  Call Extruder(294.14489)
  MoveL 3985 to (558.92, 479.39, 68) mm, rotated rx 180 ry 0 rz 160 deg; joints [3.193, 77.828, -27.011, -151.068, 54.497, 162.203]
  Set speed (17.7 mm/s)
  Call Extruder(298.39452)
  MoveL 3986 to (559.34, 480.66, 68) mm, rotated rx 180 ry 0 rz 160 deg; joints [3.332, 77.936, -27.236, -150.865, 54.438, 162.039]
  Set speed (17.7 mm/s)
  Call Extruder(302.35866)
  MoveL 3987 to (559.73, 481.84, 68) mm, rotated rx 180 ry 0 rz 160 deg; joints [3.463, 78.036, -27.442, -150.675, 54.385, 161.886]
  Call Extruder(306.52683)
  MoveL 3988 to (560.09, 483.1, 68) mm, rotated rx -180 ry 0 rz 160 deg; joints [3.601, 78.133, -27.644, -150.477, 54.338, 161.729]
  Set speed (17.7 mm/s)
  Call Extruder(310.60092)
  MoveL 3989 to (560.43, 484.33, 68) mm, rotated rx 180 ry 0 rz 160 deg; joints [3.736, 78.225, -27.836, -150.283, 54.294, 161.576]
  Set speed (17.7 mm/s)
  Call Extruder(318.62879)
  MoveL 3990 to (561.01, 486.78, 68) mm, rotated rx -180 ry 0 rz 160 deg; joints [4.006, 78.393, -28.184, -149.903, 54.224, 161.281]
  Set speed (17.7 mm/s)
  Call Extruder(326.84459)
  MoveL 3991 to (561.5, 489.31, 68) mm, rotated rx 180 ry 0 rz 160 deg; joints [4.285, 78.545, -28.498, -149.519, 54.173, 160.99]
  Set speed (17.7 mm/s)
  Call Extruder(334.91481)
  MoveL 3992 to (561.89, 491.82, 68) mm, rotated rx -180 ry 0 rz 160 deg; joints [4.561, 78.676, -28.769, -149.146, 54.144, 160.714]
  Set speed (17.7 mm/s)
  Call Extruder(343.20136)
  MoveL 3993 to (562.17, 494.4, 68) mm, rotated rx -180 ry 0 rz 160 deg; joints [4.846, 78.79, -29.004, -148.769, 54.134, 160.442]
  Set speed (17.7 mm/s)
  Call Extruder(351.25389)
  MoveL 3994 to (562.35, 496.93, 68) mm, rotated rx 180 ry 0 rz 160 deg; joints [5.124, 78.88, -29.191, -148.409, 54.146, 160.191]
  Set speed (17.7 mm/s)
  Call Extruder(359.37485)
  MoveL 3995 to (562.42, 499.47, 68) mm, rotated rx -180 ry 0 rz 160 deg; joints [5.407, 78.951, -29.336, -148.053, 54.178, 159.95]
  Set speed (17.7 mm/s)
  Call Extruder(367.60614)
  MoveL 3996 to (562.39, 502.06, 68) mm, rotated rx -180 ry 0 rz 160 deg; joints [5.694, 79.001, -29.441, -147.701, 54.232, 159.721]
  Set speed (17.7 mm/s)
  Call Extruder(375.64241)
  MoveL 3997 to (562.26, 504.58, 68) mm, rotated rx 180 ry 0 rz 160 deg; joints [5.975, 79.03, -29.501, -147.364, 54.304, 159.511]
  Set speed (17.7 mm/s)
  Call Extruder(383.68912)
  MoveL 3998 to (562.02, 507.09, 68) mm, rotated rx 180 ry 0 rz 160 deg; joints [6.256, 79.038, -29.516, -147.037, 54.396, 159.317]
  Set speed (17.7 mm/s)
  Call Extruder(391.74017)
  MoveL 3999 to (561.68, 509.6, 68) mm, rotated rx 180 ry 0 rz 160 deg; joints [6.538, 79.024, -29.487, -146.719, 54.508, 159.138]
  Set speed (17.7 mm/s)
  Call Extruder(400.03241)
  MoveL 4000 to (561.23, 512.16, 68) mm, rotated rx -180 ry 0 rz 160 deg; joints [6.827, 78.989, -29.416, -146.402, 54.643, 158.971]
  Set speed (17.7 mm/s)
  Call Extruder(408.22270)
  MoveL 4001 to (560.67, 514.68, 68) mm, rotated rx 180 ry 0 rz 160 deg; joints [7.113, 78.932, -29.298, -146.099, 54.796, 158.824]
  Set speed (17.7 mm/s)
  Call Extruder(412.26719)
  MoveL 4002 to (560.36, 515.9, 68) mm, rotated rx -180 ry 0 rz 160 deg; joints [7.253, 78.895, -29.222, -145.955, 54.879, 158.758]
  Set speed (17.7 mm/s)
  Call Extruder(416.24101)
  MoveL 4003 to (560.03, 517.11, 68) mm, rotated rx -180 ry 0 rz 160 deg; joints [7.391, 78.857, -29.142, -145.814, 54.963, 158.696]
  Set speed (17.7 mm/s)
  Call Extruder(420.44181)
  MoveL 4004 to (559.65, 518.37, 68) mm, rotated rx -180 ry 0 rz 160 deg; joints [7.536, 78.808, -29.042, -145.67, 55.059, 158.638]
  Call Extruder(424.29152)
  MoveL 4005 to (559.29, 519.52, 68) mm, rotated rx -180 ry 0 rz 160 deg; joints [7.668, 78.761, -28.945, -145.539, 55.148, 158.586]
  Set speed (17.7 mm/s)
  Call Extruder(432.46928)
  MoveL 4006 to (558.44, 521.94, 68) mm, rotated rx -180 ry 0 rz 160 deg; joints [7.949, 78.644, -28.701, -145.27, 55.354, 158.491]
  Set speed (17.7 mm/s)
  Call Extruder(436.67674)
  MoveL 4007 to (557.96, 523.17, 68) mm, rotated rx 180 ry 0 rz 160 deg; joints [8.093, 78.574, -28.558, -145.137, 55.468, 158.451]
  Set speed (17.7 mm/s)
  Call Extruder(440.85646)
  MoveL 4008 to (557.47, 524.38, 68) mm, rotated rx 180 ry 0 rz 160 deg; joints [8.235, 78.503, -28.41, -145.007, 55.583, 158.413]
  Set speed (17.7 mm/s)
  Call Extruder(448.69676)
  MoveL 4009 to (556.46, 526.63, 68) mm, rotated rx 180 ry 0 rz 160 deg; joints [8.5, 78.352, -28.098, -144.771, 55.812, 158.357]
  Set speed (17.7 mm/s)
  Call Extruder(451.96551)
  MoveL 4010 to (556.02, 527.56, 68) mm, rotated rx 180 ry 0 rz 160 deg; joints [8.61, 78.285, -27.959, -144.676, 55.912, 158.338]
  Set speed (17.7 mm/s)
  Call Extruder(459.02585)
  MoveL 4011 to (555, 529.53, 68) mm, rotated rx -180 ry 0 rz 160 deg; joints [8.846, 78.128, -27.634, -144.477, 56.136, 158.307]
  Set speed (17.7 mm/s)
  Call Extruder(465.05663)
  MoveL 4012 to (554.08, 531.18, 68) mm, rotated rx -180 ry 0 rz 160 deg; joints [9.046, 77.983, -27.333, -144.315, 56.337, 158.293]
  Set speed (17.7 mm/s)
  Call Extruder(469.10106)
  MoveL 4013 to (553.43, 532.28, 68) mm, rotated rx 180 ry 0 rz 160 deg; joints [9.179, 77.881, -27.121, -144.209, 56.475, 158.288]
  Set speed (17.7 mm/s)
  Call Extruder(472.62067)
  MoveL 4014 to (552.85, 533.22, 68) mm, rotated rx -180 ry 0 rz 160 deg; joints [9.294, 77.788, -26.929, -144.12, 56.598, 158.287]
  Set speed (17.7 mm/s)
  Call Extruder(477.24876)
  MoveL 4015 to (552.07, 534.44, 68) mm, rotated rx -180 ry 0 rz 160 deg; joints [9.444, 77.662, -26.667, -144.005, 56.764, 158.291]
  Set speed (17.7 mm/s)
  Call Extruder(482.03626)
  MoveL 4016 to (551.22, 535.68, 68) mm, rotated rx -180 ry 0 rz 160 deg; joints [9.598, 77.526, -26.384, -143.89, 56.94, 158.3]
  Set speed (17.7 mm/s)
  Call Extruder(485.47775)
  MoveL 4017 to (550.6, 536.56, 68) mm, rotated rx 180 ry 0 rz 160 deg; joints [9.708, 77.426, -26.175, -143.81, 57.068, 158.31]
  Call Extruder(489.58215)
  MoveL 4018 to (549.83, 537.6, 68) mm, rotated rx -180 ry 0 rz 160 deg; joints [9.838, 77.301, -25.915, -143.718, 57.225, 158.327]
  Call Extruder(493.57157)
  MoveL 4019 to (549.07, 538.59, 68) mm, rotated rx 180 ry 0 rz 160 deg; joints [9.964, 77.176, -25.655, -143.631, 57.38, 158.348]
  Call Extruder(497.29229)
  MoveL 4020 to (548.34, 539.5, 68) mm, rotated rx 180 ry 0 rz 160 deg; joints [10.08, 77.058, -25.408, -143.551, 57.527, 158.369]
  Set speed (17.7 mm/s)
  Call Extruder(501.66302)
  MoveL 4021 to (547.45, 540.56, 68) mm, rotated rx -180 ry 0 rz 160 deg; joints [10.215, 76.914, -25.108, -143.462, 57.702, 158.4]
  Set speed (17.7 mm/s)
  Call Extruder(505.72359)
  MoveL 4022 to (546.62, 541.52, 68) mm, rotated rx -180 ry 0 rz 160 deg; joints [10.339, 76.777, -24.821, -143.381, 57.868, 158.432]
  Call Extruder(509.84035)
  MoveL 4023 to (545.75, 542.47, 68) mm, rotated rx -180 ry 0 rz 160 deg; joints [10.464, 76.634, -24.524, -143.302, 58.038, 158.469]
  Call Extruder(513.86834)
  MoveL 4024 to (544.88, 543.39, 68) mm, rotated rx 180 ry 0 rz 160 deg; joints [10.585, 76.492, -24.226, -143.227, 58.207, 158.508]
  Call Extruder(517.98050)
  MoveL 4025 to (543.97, 544.31, 68) mm, rotated rx 180 ry 0 rz 160 deg; joints [10.707, 76.343, -23.915, -143.154, 58.382, 158.553]
  Set speed (17.7 mm/s)
  Call Extruder(522.01486)
  MoveL 4026 to (543.06, 545.19, 68) mm, rotated rx -180 ry 0 rz 160 deg; joints [10.826, 76.194, -23.602, -143.085, 58.556, 158.6]
  Set speed (17.7 mm/s)
  Call Extruder(526.03664)
  MoveL 4027 to (542.14, 546.05, 68) mm, rotated rx -180 ry 0 rz 160 deg; joints [10.942, 76.043, -23.286, -143.018, 58.731, 158.65]
  Set speed (17.7 mm/s)
  Call Extruder(530.16740)
  MoveL 4028 to (541.17, 546.92, 68) mm, rotated rx 180 ry 0 rz 160 deg; joints [11.061, 75.885, -22.954, -142.953, 58.913, 158.706]
  Set speed (17.7 mm/s)
  Call Extruder(534.20745)
  MoveL 4029 to (540.21, 547.75, 68) mm, rotated rx 180 ry 0 rz 160 deg; joints [11.175, 75.728, -22.623, -142.891, 59.092, 158.764]
  Call Extruder(538.24993)
  MoveL 4030 to (539.23, 548.55, 68) mm, rotated rx -180 ry 0 rz 160 deg; joints [11.288, 75.568, -22.286, -142.832, 59.274, 158.825]
  Set speed (17.7 mm/s)
  Call Extruder(542.31774)
  MoveL 4031 to (538.23, 549.35, 68) mm, rotated rx 180 ry 0 rz 160 deg; joints [11.4, 75.404, -21.942, -142.775, 59.459, 158.89]
  Set speed (17.7 mm/s)
  Call Extruder(546.38760)
  MoveL 4032 to (537.21, 550.12, 68) mm, rotated rx 180 ry 0 rz 160 deg; joints [11.511, 75.238, -21.592, -142.721, 59.645, 158.959]
  Set speed (17.7 mm/s)
  Call Extruder(550.65806)
  MoveL 4033 to (536.13, 550.91, 68) mm, rotated rx -180 ry 0 rz 160 deg; joints [11.625, 75.062, -21.22, -142.667, 59.842, 159.034]
  Call Extruder(554.55663)
  MoveL 4034 to (535.12, 551.61, 68) mm, rotated rx 180 ry 0 rz 160 deg; joints [11.728, 74.899, -20.875, -142.619, 60.023, 159.106]
  Set speed (17.7 mm/s)
  Call Extruder(558.59833)
  MoveL 4035 to (534.07, 552.31, 68) mm, rotated rx 180 ry 0 rz 160 deg; joints [11.833, 74.727, -20.512, -142.573, 60.212, 159.184]
  Set speed (17.7 mm/s)
  Call Extruder(562.67182)
  MoveL 4036 to (532.99, 553, 68) mm, rotated rx 180 ry 0 rz 160 deg; joints [11.937, 74.552, -20.142, -142.529, 60.404, 159.265]
  Set speed (17.7 mm/s)
  Call Extruder(566.75852)
  MoveL 4037 to (531.89, 553.66, 68) mm, rotated rx 180 ry 0 rz 160 deg; joints [12.039, 74.375, -19.767, -142.488, 60.597, 159.349]
  Set speed (17.7 mm/s)
  Call Extruder(570.85954)
  MoveL 4038 to (530.78, 554.31, 68) mm, rotated rx -180 ry 0 rz 160 deg; joints [12.14, 74.196, -19.386, -142.448, 60.793, 159.437]
  Set speed (17.7 mm/s)
  Call Extruder(576.98550)
  MoveL 4039 to (529.09, 555.24, 68) mm, rotated rx -180 ry 0 rz 160 deg; joints [12.288, 73.925, -18.81, -142.393, 61.086, 159.573]
  Call Extruder(583.05688)
  MoveL 4040 to (527.39, 556.1, 68) mm, rotated rx 180 ry 0 rz 160 deg; joints [12.429, 73.652, -18.229, -142.346, 61.379, 159.715]
  Set speed (17.7 mm/s)
  Call Extruder(587.00755)
  MoveL 4041 to (526.27, 556.63, 68) mm, rotated rx -180 ry 0 rz 160 deg; joints [12.519, 73.473, -17.847, -142.317, 61.571, 159.81]
  Set speed (17.7 mm/s)
  Call Extruder(591.18449)
  MoveL 4042 to (525.07, 557.16, 68) mm, rotated rx -180 ry 0 rz 160 deg; joints [12.61, 73.282, -17.44, -142.29, 61.774, 159.914]
  Set speed (17.7 mm/s)
  Call Extruder(595.25468)
  MoveL 4043 to (523.9, 557.67, 68) mm, rotated rx -180 ry 0 rz 160 deg; joints [12.699, 73.096, -17.042, -142.265, 61.971, 160.016]
  Call Extruder(599.32932)
  MoveL 4044 to (522.71, 558.14, 68) mm, rotated rx 180 ry 0 rz 160 deg; joints [12.784, 72.908, -16.639, -142.244, 62.17, 160.123]
  Set speed (17.7 mm/s)
  Call Extruder(603.41760)
  MoveL 4045 to (521.51, 558.6, 68) mm, rotated rx -180 ry 0 rz 160 deg; joints [12.869, 72.719, -16.234, -142.224, 62.37, 160.231]
  Set speed (17.7 mm/s)
  Call Extruder(607.51619)
  MoveL 4046 to (520.3, 559.02, 68) mm, rotated rx 180 ry 0 rz 160 deg; joints [12.95, 72.527, -15.823, -142.208, 62.571, 160.342]
  Set speed (17.7 mm/s)
  Call Extruder(611.50972)
  MoveL 4047 to (519.11, 559.43, 68) mm, rotated rx 180 ry 0 rz 160 deg; joints [13.029, 72.341, -15.423, -142.192, 62.766, 160.452]
  Set speed (17.7 mm/s)
  Call Extruder(615.60966)
  MoveL 4048 to (517.88, 559.8, 68) mm, rotated rx -180 ry 0 rz 160 deg; joints [13.105, 72.148, -15.007, -142.181, 62.968, 160.568]
  Call Extruder(619.63022)
  MoveL 4049 to (516.67, 560.16, 68) mm, rotated rx 180 ry 0 rz 160 deg; joints [13.18, 71.959, -14.6, -142.171, 63.165, 160.683]
  Set speed (17.7 mm/s)
  Call Extruder(623.21774)
  MoveL 4050 to (515.59, 560.44, 68) mm, rotated rx -180 ry 0 rz 160 deg; joints [13.243, 71.79, -14.233, -142.165, 63.341, 160.788]
  Call Extruder(627.77646)
  MoveL 4051 to (514.2, 560.79, 68) mm, rotated rx -180 ry 0 rz 160 deg; joints [13.321, 71.574, -13.768, -142.158, 63.564, 160.922]
  Set speed (17.7 mm/s)
  Call Extruder(635.96464)
  MoveL 4052 to (511.68, 561.32, 68) mm, rotated rx 180 ry 0 rz 160 deg; joints [13.454, 71.185, -12.924, -142.156, 63.966, 161.171]
  Set speed (17.7 mm/s)
  Call Extruder(644.15315)
  MoveL 4053 to (509.15, 561.75, 68) mm, rotated rx 180 ry 0 rz 160 deg; joints [13.576, 70.795, -12.077, -142.163, 64.367, 161.427]
  Set speed (17.7 mm/s)
  Call Extruder(652.20654)
  MoveL 4054 to (506.64, 562.07, 68) mm, rotated rx 180 ry 0 rz 160 deg; joints [13.686, 70.411, -11.24, -142.179, 64.759, 161.685]
  Set speed (17.7 mm/s)
  Call Extruder(660.39241)
  MoveL 4055 to (504.08, 562.29, 68) mm, rotated rx -180 ry 0 rz 160 deg; joints [13.787, 70.021, -10.386, -142.207, 65.157, 161.954]
  Set speed (17.7 mm/s)
  Call Extruder(668.57383)
  MoveL 4056 to (501.52, 562.4, 68) mm, rotated rx 180 ry 0 rz 160 deg; joints [13.876, 69.632, -9.533, -142.244, 65.551, 162.228]
  Set speed (17.7 mm/s)
  Call Extruder(676.52907)
  MoveL 4057 to (499.02, 562.42, 68) mm, rotated rx 180 ry 0 rz 160 deg; joints [13.952, 69.256, -8.704, -142.289, 65.932, 162.499]
  Set speed (10.0 mm/s)
  MoveL 4058 to (499.02, 562.42, 72) mm, rotated rx 180 ry 0 rz 160 deg; joints [13.952, 68.584, -8.319, -142.211, 65.706, 162.307]
  Set speed (120.0 mm/s)
  MoveL 4059 to (498.98, 563.11, 72) mm, rotated rx 180 ry 0 rz 160 deg; joints [14.037, 68.604, -8.362, -142.116, 65.713, 162.255]
  Set speed (17.8 mm/s)
  Call Extruder(684.78584)
  MoveL 4060 to (496.38, 563.01, 72) mm, rotated rx 180 ry 0 rz 160 deg; joints [14.103, 68.213, -7.503, -142.174, 66.103, 162.541]
  Set speed (17.7 mm/s)
  Call Extruder(693.01751)
  MoveL 4061 to (493.8, 562.81, 72) mm, rotated rx 180 ry 0 rz 160 deg; joints [14.158, 67.826, -6.651, -142.243, 66.487, 162.83]
  Set speed (17.8 mm/s)
  Call Extruder(701.15810)
  MoveL 4062 to (491.26, 562.51, 72) mm, rotated rx 180 ry 0 rz 160 deg; joints [14.199, 67.447, -5.811, -142.321, 66.863, 163.119]
  Set speed (17.8 mm/s)
  Call Extruder(709.32825)
  MoveL 4063 to (488.72, 562.1, 72) mm, rotated rx 180 ry 0 rz 160 deg; joints [14.228, 67.07, -4.974, -142.411, 67.236, 163.413]
  Call Extruder(717.38257)
  MoveL 4064 to (486.24, 561.6, 72) mm, rotated rx -180 ry 0 rz 160 deg; joints [14.243, 66.702, -4.155, -142.509, 67.598, 163.705]
  Set speed (17.7 mm/s)
  Call Extruder(721.73346)
  MoveL 4065 to (484.9, 561.28, 72) mm, rotated rx 180 ry 0 rz 160 deg; joints [14.246, 66.506, -3.716, -142.567, 67.791, 163.863]
  Set speed (17.7 mm/s)
  Call Extruder(725.73905)
  MoveL 4066 to (483.69, 560.97, 72) mm, rotated rx -180 ry 0 rz 160 deg; joints [14.246, 66.326, -3.314, -142.621, 67.968, 164.008]
  Call Extruder(729.90744)
  MoveL 4067 to (482.43, 560.62, 72) mm, rotated rx 180 ry 0 rz 160 deg; joints [14.242, 66.14, -2.898, -142.682, 68.15, 164.161]
  Set speed (17.7 mm/s)
  Call Extruder(734.10375)
  MoveL 4068 to (481.16, 560.24, 72) mm, rotated rx 180 ry 0 rz 160 deg; joints [14.235, 65.955, -2.481, -142.745, 68.332, 164.314]
  Set speed (17.7 mm/s)
  Call Extruder(738.10997)
  MoveL 4069 to (479.97, 559.85, 72) mm, rotated rx 180 ry 0 rz 160 deg; joints [14.223, 65.779, -2.086, -142.809, 68.504, 164.462]
  Set speed (17.7 mm/s)
  Call Extruder(742.27099)
  MoveL 4070 to (478.73, 559.43, 72) mm, rotated rx 180 ry 0 rz 160 deg; joints [14.21, 65.598, -1.678, -142.877, 68.681, 164.614]
  Set speed (17.7 mm/s)
  Call Extruder(746.37719)
  MoveL 4071 to (477.52, 558.97, 72) mm, rotated rx 180 ry 0 rz 160 deg; joints [14.191, 65.421, -1.278, -142.949, 68.854, 164.765]
  Call Extruder(750.35027)
  MoveL 4072 to (476.36, 558.52, 72) mm, rotated rx 180 ry 0 rz 160 deg; joints [14.172, 65.251, -0.893, -143.019, 69.02, 164.911]
  Set speed (17.7 mm/s)
  Call Extruder(752.50038)
  MoveL 4073 to (475.73, 558.27, 72) mm, rotated rx 180 ry 0 rz 160 deg; joints [14.159, 65.16, -0.687, -143.058, 69.109, 164.99]
  Set speed (17.7 mm/s)
  Call Extruder(758.47349)
  MoveL 4074 to (474.01, 557.52, 72) mm, rotated rx 180 ry 0 rz 160 deg; joints [14.119, 64.909, -0.117, -143.172, 69.354, 165.209]
  Set speed (17.8 mm/s)
  Call Extruder(762.73063)
  MoveL 4075 to (472.8, 556.95, 72) mm, rotated rx -180 ry 0 rz 160 deg; joints [14.086, 64.732, 0.286, -143.257, 69.527, 165.366]
  Call Extruder(766.79294)
  MoveL 4076 to (471.65, 556.39, 72) mm, rotated rx 180 ry 0 rz 160 deg; joints [14.051, 64.565, 0.667, -143.341, 69.689, 165.515]
  Set speed (17.7 mm/s)
  Call Extruder(769.82727)
  MoveL 4077 to (470.8, 555.96, 72) mm, rotated rx -180 ry 0 rz 160 deg; joints [14.023, 64.442, 0.949, -143.405, 69.81, 165.626]
  Set speed (17.7 mm/s)
  Call Extruder(775.14653)
  MoveL 4078 to (469.33, 555.16, 72) mm, rotated rx 180 ry 0 rz 160 deg; joints [13.968, 64.228, 1.439, -143.522, 70.018, 165.82]
  Set speed (17.8 mm/s)
  Call Extruder(779.12231)
  MoveL 4079 to (468.24, 554.54, 72) mm, rotated rx 180 ry 0 rz 160 deg; joints [13.923, 64.07, 1.801, -143.612, 70.171, 165.965]
  Set speed (17.8 mm/s)
  Call Extruder(783.32191)
  MoveL 4080 to (467.11, 553.87, 72) mm, rotated rx -180 ry 0 rz 160 deg; joints [13.871, 63.905, 2.18, -143.711, 70.331, 166.118]
  Set speed (17.8 mm/s)
  Call Extruder(787.31436)
  MoveL 4081 to (466.04, 553.2, 72) mm, rotated rx 180 ry 0 rz 160 deg; joints [13.819, 63.75, 2.536, -143.807, 70.481, 166.262]
  Set speed (17.8 mm/s)
  Call Extruder(791.45586)
  MoveL 4082 to (464.95, 552.49, 72) mm, rotated rx -180 ry 0 rz 160 deg; joints [13.761, 63.592, 2.901, -143.91, 70.634, 166.411]
  Set speed (17.8 mm/s)
  Call Extruder(795.56231)
  MoveL 4083 to (463.88, 551.76, 72) mm, rotated rx -180 ry 0 rz 160 deg; joints [13.7, 63.437, 3.259, -144.015, 70.784, 166.559]
  Set speed (17.8 mm/s)
  Call Extruder(799.66580)
  MoveL 4084 to (462.83, 551.01, 72) mm, rotated rx -180 ry 0 rz 160 deg; joints [13.635, 63.285, 3.613, -144.122, 70.932, 166.705]
  Set speed (17.7 mm/s)
  Call Extruder(803.84529)
  MoveL 4085 to (461.78, 550.23, 72) mm, rotated rx -180 ry 0 rz 160 deg; joints [13.566, 63.132, 3.968, -144.235, 71.08, 166.854]
  Set speed (17.7 mm/s)
  Call Extruder(807.89672)
  MoveL 4086 to (460.77, 549.45, 72) mm, rotated rx 180 ry 0 rz 160 deg; joints [13.494, 62.986, 4.308, -144.346, 71.221, 166.997]
  Set speed (17.8 mm/s)
  Call Extruder(812.15374)
  MoveL 4087 to (459.73, 548.6, 72) mm, rotated rx 180 ry 0 rz 160 deg; joints [13.416, 62.834, 4.66, -144.467, 71.367, 167.146]
  Call Extruder(816.08698)
  MoveL 4088 to (458.79, 547.8, 72) mm, rotated rx 180 ry 0 rz 160 deg; joints [13.339, 62.697, 4.98, -144.581, 71.499, 167.284]
  Call Extruder(820.12043)
  MoveL 4089 to (457.83, 546.96, 72) mm, rotated rx -180 ry 0 rz 160 deg; joints [13.258, 62.558, 5.305, -144.701, 71.633, 167.423]
  Set speed (17.8 mm/s)
  Call Extruder(824.28360)
  MoveL 4090 to (456.87, 546.08, 72) mm, rotated rx 180 ry 0 rz 160 deg; joints [13.17, 62.418, 5.634, -144.827, 71.768, 167.567]
  Set speed (17.8 mm/s)
  Call Extruder(828.39151)
  MoveL 4091 to (455.93, 545.19, 72) mm, rotated rx 180 ry 0 rz 160 deg; joints [13.079, 62.282, 5.954, -144.955, 71.899, 167.707]
  Call Extruder(832.47818)
  MoveL 4092 to (455.02, 544.28, 72) mm, rotated rx -180 ry 0 rz 160 deg; joints [12.986, 62.149, 6.267, -145.085, 72.027, 167.845]
  Set speed (17.8 mm/s)
  Call Extruder(836.60977)
  MoveL 4093 to (454.12, 543.34, 72) mm, rotated rx -180 ry 0 rz 160 deg; joints [12.888, 62.017, 6.578, -145.219, 72.153, 167.983]
  Set speed (17.8 mm/s)
  Call Extruder(840.62722)
  MoveL 4094 to (453.26, 542.42, 72) mm, rotated rx 180 ry 0 rz 160 deg; joints [12.789, 61.891, 6.875, -145.351, 72.273, 168.117]
  Call Extruder(844.81137)
  MoveL 4095 to (452.39, 541.43, 72) mm, rotated rx -180 ry 0 rz 160 deg; joints [12.682, 61.763, 7.178, -145.493, 72.396, 168.255]
  Call Extruder(848.43498)
  MoveL 4096 to (451.65, 540.57, 72) mm, rotated rx -180 ry 0 rz 160 deg; joints [12.587, 61.654, 7.436, -145.617, 72.499, 168.373]
  Set speed (17.8 mm/s)
  Call Extruder(853.01287)
  MoveL 4097 to (450.73, 539.45, 72) mm, rotated rx -180 ry 0 rz 160 deg; joints [12.463, 61.519, 7.756, -145.778, 72.627, 168.52]
  Call Extruder(857.11960)
  MoveL 4098 to (449.94, 538.43, 72) mm, rotated rx 180 ry 0 rz 160 deg; joints [12.348, 61.402, 8.036, -145.924, 72.739, 168.651]
  Set speed (17.8 mm/s)
  Call Extruder(861.20079)
  MoveL 4099 to (449.16, 537.41, 72) mm, rotated rx 180 ry 0 rz 160 deg; joints [12.23, 61.287, 8.309, -146.072, 72.847, 168.779]
  Call Extruder(865.32794)
  MoveL 4100 to (448.4, 536.36, 72) mm, rotated rx 180 ry 0 rz 160 deg; joints [12.108, 61.174, 8.578, -146.225, 72.954, 168.907]
  Call Extruder(869.40800)
  MoveL 4101 to (447.68, 535.3, 72) mm, rotated rx 180 ry 0 rz 160 deg; joints [11.983, 61.065, 8.838, -146.378, 73.056, 169.033]
  Set speed (17.8 mm/s)
  Call Extruder(873.51158)
  MoveL 4102 to (446.97, 534.22, 72) mm, rotated rx 180 ry 0 rz 160 deg; joints [11.855, 60.959, 9.094, -146.535, 73.156, 169.157]
  Set speed (17.8 mm/s)
  Call Extruder(877.62154)
  MoveL 4103 to (446.27, 533.13, 72) mm, rotated rx 180 ry 0 rz 160 deg; joints [11.723, 60.855, 9.344, -146.694, 73.253, 169.279]
  Set speed (17.8 mm/s)
  Call Extruder(881.67014)
  MoveL 4104 to (445.62, 532.04, 72) mm, rotated rx -180 ry 0 rz 160 deg; joints [11.591, 60.755, 9.583, -146.853, 73.345, 169.399]
  Call Extruder(885.83166)
  MoveL 4105 to (444.96, 530.9, 72) mm, rotated rx -180 ry 0 rz 160 deg; joints [11.451, 60.656, 9.822, -147.019, 73.437, 169.519]
  Call Extruder(889.93873)
  MoveL 4106 to (444.35, 529.77, 72) mm, rotated rx 180 ry 0 rz 160 deg; joints [11.31, 60.561, 10.051, -147.186, 73.524, 169.636]
  Call Extruder(894.04948)
  MoveL 4107 to (443.75, 528.62, 72) mm, rotated rx 180 ry 0 rz 160 deg; joints [11.166, 60.469, 10.274, -147.354, 73.608, 169.752]
  Set speed (17.8 mm/s)
  Call Extruder(898.06498)
  MoveL 4108 to (443.18, 527.49, 72) mm, rotated rx -180 ry 0 rz 160 deg; joints [11.022, 60.382, 10.485, -147.521, 73.687, 169.862]
  Set speed (17.7 mm/s)
  Call Extruder(902.33645)
  MoveL 4109 to (442.62, 526.27, 72) mm, rotated rx -180 ry 0 rz 160 deg; joints [10.866, 60.293, 10.7, -147.701, 73.766, 169.978]
  Set speed (17.7 mm/s)
  Call Extruder(906.43110)
  MoveL 4110 to (442.09, 525.1, 72) mm, rotated rx -180 ry 0 rz 160 deg; joints [10.715, 60.21, 10.902, -147.874, 73.84, 170.087]
  Set speed (17.7 mm/s)
  Call Extruder(910.55447)
  MoveL 4111 to (441.59, 523.9, 72) mm, rotated rx -180 ry 0 rz 160 deg; joints [10.559, 60.13, 11.096, -148.052, 73.91, 170.194]
  Set speed (17.7 mm/s)
  Call Extruder(914.45439)
  MoveL 4112 to (441.13, 522.77, 72) mm, rotated rx 180 ry 0 rz 160 deg; joints [10.41, 60.057, 11.274, -148.221, 73.975, 170.295]
  Set speed (17.7 mm/s)
  Call Extruder(918.77421)
  MoveL 4113 to (440.66, 521.5, 72) mm, rotated rx -180 ry 0 rz 160 deg; joints [10.241, 59.98, 11.462, -148.41, 74.04, 170.403]
  Call Extruder(922.87536)
  MoveL 4114 to (440.23, 520.28, 72) mm, rotated rx 180 ry 0 rz 160 deg; joints [10.08, 59.908, 11.636, -148.591, 74.101, 170.504]
  Set speed (17.8 mm/s)
  Call Extruder(931.08749)
  MoveL 4115 to (439.45, 517.82, 72) mm, rotated rx 180 ry 0 rz 160 deg; joints [9.747, 59.777, 11.958, -148.96, 74.21, 170.7]
  Set speed (17.7 mm/s)
  Call Extruder(935.19094)
  MoveL 4116 to (439.11, 516.58, 72) mm, rotated rx 180 ry 0 rz 160 deg; joints [9.578, 59.716, 12.106, -149.147, 74.257, 170.794]
  Set speed (17.7 mm/s)
  Call Extruder(939.16372)
  MoveL 4117 to (438.79, 515.37, 72) mm, rotated rx 180 ry 0 rz 160 deg; joints [9.412, 59.66, 12.245, -149.328, 74.302, 170.883]
  Set speed (17.7 mm/s)
  Call Extruder(943.40434)
  MoveL 4118 to (438.48, 514.07, 72) mm, rotated rx 180 ry 0 rz 160 deg; joints [9.233, 59.604, 12.382, -149.524, 74.344, 170.976]
  Call Extruder(947.41026)
  MoveL 4119 to (438.2, 512.85, 72) mm, rotated rx 180 ry 0 rz 160 deg; joints [9.062, 59.552, 12.508, -149.71, 74.381, 171.062]
  Set speed (17.8 mm/s)
  Call Extruder(955.74907)
  MoveL 4120 to (437.72, 510.27, 72) mm, rotated rx -180 ry 0 rz 160 deg; joints [8.701, 59.457, 12.742, -150.1, 74.446, 171.234]
  Set speed (17.7 mm/s)
  Call Extruder(963.95051)
  MoveL 4121 to (437.36, 507.71, 72) mm, rotated rx 180 ry 0 rz 160 deg; joints [8.339, 59.377, 12.94, -150.487, 74.494, 171.394]
  Call Extruder(972.16130)
  MoveL 4122 to (437.1, 505.15, 72) mm, rotated rx 180 ry 0 rz 160 deg; joints [7.971, 59.309, 13.107, -150.878, 74.526, 171.546]
  Call Extruder(980.19898)
  MoveL 4123 to (436.94, 502.62, 72) mm, rotated rx 180 ry 0 rz 160 deg; joints [7.607, 59.255, 13.24, -151.263, 74.542, 171.685]
  Set speed (17.7 mm/s)
  Call Extruder(988.50118)
  MoveL 4124 to (436.88, 500.01, 72) mm, rotated rx 180 ry 0 rz 160 deg; joints [7.227, 59.213, 13.344, -151.661, 74.542, 171.82]
  Call Extruder(995.96639)
  MoveL 4125 to (436.93, 497.66, 72) mm, rotated rx -180 ry 0 rz 160 deg; joints [6.883, 59.187, 13.41, -152.019, 74.528, 171.933]
  Call Extruder(1003.17441)
  MoveL 4126 to (437.05, 495.4, 72) mm, rotated rx 180 ry 0 rz 160 deg; joints [6.55, 59.172, 13.447, -152.364, 74.501, 172.035]
  Call Extruder(1010.66998)
  MoveL 4127 to (437.27, 493.06, 72) mm, rotated rx 180 ry 0 rz 160 deg; joints [6.203, 59.167, 13.459, -152.722, 74.459, 172.134]
  Call Extruder(1018.05787)
  MoveL 4128 to (437.56, 490.75, 72) mm, rotated rx -180 ry 0 rz 160 deg; joints [5.861, 59.173, 13.445, -153.073, 74.405, 172.225]
  Set speed (17.7 mm/s)
  Call Extruder(1025.53388)
  MoveL 4129 to (437.95, 488.43, 72) mm, rotated rx 180 ry 0 rz 160 deg; joints [5.515, 59.189, 13.403, -153.425, 74.337, 172.309]
  Set speed (17.8 mm/s)
  Call Extruder(1032.83144)
  MoveL 4130 to (438.41, 486.18, 72) mm, rotated rx 180 ry 0 rz 160 deg; joints [5.179, 59.216, 13.337, -153.766, 74.257, 172.384]
  Call Extruder(1040.21403)
  MoveL 4131 to (438.96, 483.93, 72) mm, rotated rx 180 ry 0 rz 160 deg; joints [4.841, 59.254, 13.243, -154.107, 74.162, 172.453]
  Call Extruder(1047.50290)
  MoveL 4132 to (439.59, 481.72, 72) mm, rotated rx -180 ry 0 rz 160 deg; joints [4.511, 59.302, 13.125, -154.44, 74.055, 172.515]
  Set speed (17.8 mm/s)
  Call Extruder(1054.91227)
  MoveL 4133 to (440.31, 479.5, 72) mm, rotated rx 180 ry 0 rz 160 deg; joints [4.178, 59.361, 12.979, -154.772, 73.934, 172.571]
  Set speed (17.8 mm/s)
  Call Extruder(1062.45704)
  MoveL 4134 to (441.12, 477.27, 72) mm, rotated rx 180 ry 0 rz 160 deg; joints [3.843, 59.432, 12.803, -155.105, 73.796, 172.621]
  Set speed (17.8 mm/s)
  Call Extruder(1069.84361)
  MoveL 4135 to (441.99, 475.12, 72) mm, rotated rx 180 ry 0 rz 160 deg; joints [3.521, 59.512, 12.606, -155.424, 73.648, 172.663]
  Set speed (17.8 mm/s)
  Call Extruder(1077.06733)
  MoveL 4136 to (442.93, 473.05, 72) mm, rotated rx 180 ry 0 rz 160 deg; joints [3.211, 59.601, 12.389, -155.728, 73.491, 172.698]
  Set speed (17.8 mm/s)
  Call Extruder(1084.52838)
  MoveL 4137 to (443.97, 470.94, 72) mm, rotated rx 180 ry 0 rz 160 deg; joints [2.897, 59.703, 12.139, -156.035, 73.316, 172.728]
  Set speed (17.7 mm/s)
  Call Extruder(1091.84400)
  MoveL 4138 to (445.07, 468.92, 72) mm, rotated rx -180 ry 0 rz 160 deg; joints [2.595, 59.813, 11.87, -156.328, 73.132, 172.751]
  Call Extruder(1099.24095)
  MoveL 4139 to (446.25, 466.92, 72) mm, rotated rx 180 ry 0 rz 160 deg; joints [2.298, 59.934, 11.573, -156.615, 72.934, 172.768]
  Set speed (17.8 mm/s)
  Call Extruder(1106.68812)
  MoveL 4140 to (447.51, 464.94, 72) mm, rotated rx -180 ry 0 rz 160 deg; joints [2.006, 60.067, 11.25, -156.895, 72.722, 172.778]
  Set speed (17.8 mm/s)
  Call Extruder(1114.06686)
  MoveL 4141 to (448.84, 463.04, 72) mm, rotated rx -180 ry 0 rz 160 deg; joints [1.726, 60.208, 10.907, -157.162, 72.501, 172.783]
  Call Extruder(1121.45273)
  MoveL 4142 to (450.23, 461.18, 72) mm, rotated rx 180 ry 0 rz 160 deg; joints [1.453, 60.359, 10.539, -157.419, 72.267, 172.781]
  Set speed (17.8 mm/s)
  Call Extruder(1128.76650)
  MoveL 4143 to (451.68, 459.39, 72) mm, rotated rx 180 ry 0 rz 160 deg; joints [1.193, 60.519, 10.153, -157.663, 72.026, 172.774]
  Set speed (17.8 mm/s)
  Call Extruder(1136.30058)
  MoveL 4144 to (453.24, 457.61, 72) mm, rotated rx 180 ry 0 rz 160 deg; joints [0.934, 60.693, 9.733, -157.903, 71.765, 172.76]
  Set speed (17.8 mm/s)
  Call Extruder(1143.69286)
  MoveL 4145 to (454.83, 455.91, 72) mm, rotated rx -180 ry 0 rz 160 deg; joints [0.69, 60.874, 9.299, -158.126, 71.499, 172.74]
  Call Extruder(1150.92671)
  MoveL 4146 to (456.45, 454.31, 72) mm, rotated rx 180 ry 0 rz 160 deg; joints [0.462, 61.059, 8.853, -158.332, 71.229, 172.715]
  Set speed (17.8 mm/s)
  Call Extruder(1158.37668)
  MoveL 4147 to (458.18, 452.73, 72) mm, rotated rx 180 ry 0 rz 160 deg; joints [0.237, 61.26, 8.374, -158.533, 70.941, 172.683]
  Call Extruder(1165.83726)
  MoveL 4148 to (459.97, 451.2, 72) mm, rotated rx -180 ry 0 rz 160 deg; joints [0.023, 61.47, 7.874, -158.721, 70.644, 172.645]
  Call Extruder(1173.08996)
  MoveL 4149 to (461.76, 449.79, 72) mm, rotated rx 180 ry 0 rz 160 deg; joints [-0.175, 61.683, 7.368, -158.891, 70.345, 172.602]
  Set speed (17.8 mm/s)
  Call Extruder(1180.53960)
  MoveL 4150 to (463.65, 448.4, 72) mm, rotated rx -180 ry 0 rz 160 deg; joints [-0.366, 61.91, 6.83, -159.053, 70.031, 172.552]
  Set speed (17.8 mm/s)
  Call Extruder(1187.91519)
  MoveL 4151 to (465.57, 447.1, 72) mm, rotated rx -180 ry 0 rz 160 deg; joints [-0.544, 62.143, 6.279, -159.2, 69.711, 172.496]
  Set speed (17.8 mm/s)
  Call Extruder(1195.37483)
  MoveL 4152 to (467.56, 445.86, 72) mm, rotated rx 180 ry 0 rz 160 deg; joints [-0.713, 62.388, 5.704, -159.334, 69.38, 172.433]
  Call Extruder(1202.76870)
  MoveL 4153 to (469.58, 444.7, 72) mm, rotated rx 180 ry 0 rz 160 deg; joints [-0.868, 62.639, 5.117, -159.454, 69.044, 172.365]
  Set speed (17.8 mm/s)
  Call Extruder(1210.14744)
  MoveL 4154 to (471.63, 443.62, 72) mm, rotated rx -180 ry 0 rz 160 deg; joints [-1.011, 62.896, 4.516, -159.559, 68.703, 172.291]
  Set speed (17.7 mm/s)
  Call Extruder(1217.35488)
  MoveL 4155 to (473.68, 442.64, 72) mm, rotated rx 180 ry 0 rz 160 deg; joints [-1.139, 63.155, 3.913, -159.648, 68.364, 172.212]
  Set speed (17.7 mm/s)
  Call Extruder(1224.66217)
  MoveL 4156 to (475.78, 441.72, 72) mm, rotated rx -180 ry 0 rz 160 deg; joints [-1.257, 63.425, 3.288, -159.725, 68.014, 172.126]
  Set speed (17.8 mm/s)
  Call Extruder(1232.15640)
  MoveL 4157 to (477.97, 440.85, 72) mm, rotated rx -180 ry 0 rz 160 deg; joints [-1.366, 63.709, 2.632, -159.79, 67.65, 172.031]
  Call Extruder(1239.70404)
  MoveL 4158 to (480.21, 440.06, 72) mm, rotated rx -180 ry 0 rz 160 deg; joints [-1.464, 64.002, 1.958, -159.84, 67.279, 171.929]
  Call Extruder(1246.94387)
  MoveL 4159 to (482.39, 439.39, 72) mm, rotated rx -180 ry 0 rz 160 deg; joints [-1.546, 64.289, 1.298, -159.874, 66.918, 171.824]
  Set speed (17.8 mm/s)
  Call Extruder(1254.37889)
  MoveL 4160 to (484.65, 438.78, 72) mm, rotated rx -180 ry 0 rz 160 deg; joints [-1.619, 64.591, 0.609, -159.895, 66.543, 171.71]
  Set speed (17.8 mm/s)
  Call Extruder(1261.85377)
  MoveL 4161 to (486.94, 438.25, 72) mm, rotated rx 180 ry 0 rz 160 deg; joints [-1.68, 64.9, -0.096, -159.901, 66.163, 171.588]
  Call Extruder(1269.16307)
  MoveL 4162 to (489.2, 437.82, 72) mm, rotated rx 180 ry 0 rz 160 deg; joints [-1.728, 65.208, -0.795, -159.893, 65.789, 171.462]
  Set speed (17.8 mm/s)
  Call Extruder(1276.21705)
  MoveL 4163 to (491.39, 437.47, 72) mm, rotated rx -180 ry 0 rz 160 deg; joints [-1.764, 65.51, -1.479, -159.873, 65.425, 171.334]
  Set speed (17.8 mm/s)
  Call Extruder(1283.97093)
  MoveL 4164 to (493.81, 437.19, 72) mm, rotated rx -180 ry 0 rz 160 deg; joints [-1.791, 65.848, -2.24, -159.835, 65.023, 171.186]
  Set speed (17.8 mm/s)
  Call Extruder(1291.23915)
  MoveL 4165 to (496.09, 437.01, 72) mm, rotated rx 180 ry 0 rz 160 deg; joints [-1.805, 66.169, -2.961, -159.786, 64.645, 171.04]
  Set speed (17.8 mm/s)
  Call Extruder(1298.78214)
  MoveL 4166 to (498.46, 436.9, 72) mm, rotated rx 180 ry 0 rz 160 deg; joints [-1.809, 66.507, -3.718, -159.72, 64.252, 170.881]
  Set speed (17.8 mm/s)
  Call Extruder(1306.09276)
  MoveL 4167 to (500.76, 436.89, 72) mm, rotated rx -180 ry 0 rz 160 deg; joints [-1.801, 66.838, -4.458, -159.643, 63.87, 170.719]
  Set speed (17.8 mm/s)
  Call Extruder(1313.36661)
  MoveL 4168 to (503.05, 436.96, 72) mm, rotated rx 180 ry 0 rz 160 deg; joints [-1.784, 67.171, -5.2, -159.553, 63.49, 170.552]
  Call Extruder(1320.86065)
  MoveL 4169 to (505.41, 437.12, 72) mm, rotated rx 180 ry 0 rz 160 deg; joints [-1.754, 67.518, -5.969, -159.447, 63.099, 170.372]
  Set speed (17.8 mm/s)
  Call Extruder(1328.11823)
  MoveL 4170 to (507.68, 437.35, 72) mm, rotated rx -180 ry 0 rz 160 deg; joints [-1.716, 67.857, -6.718, -159.33, 62.722, 170.19]
  Set speed (17.7 mm/s)
  Call Extruder(1335.56301)
  MoveL 4171 to (510, 437.68, 72) mm, rotated rx 180 ry 0 rz 160 deg; joints [-1.666, 68.207, -7.489, -159.198, 62.336, 169.997]
  Set speed (17.8 mm/s)
  Call Extruder(1343.08625)
  MoveL 4172 to (512.33, 438.1, 72) mm, rotated rx -180 ry 0 rz 160 deg; joints [-1.606, 68.563, -8.271, -159.05, 61.948, 169.794]
  Set speed (17.8 mm/s)
  Call Extruder(1350.27580)
  MoveL 4173 to (514.54, 438.58, 72) mm, rotated rx -180 ry 0 rz 160 deg; joints [-1.539, 68.905, -9.02, -158.897, 61.58, 169.592]
  Set speed (17.8 mm/s)
  Call Extruder(1357.71641)
  MoveL 4174 to (516.8, 439.16, 72) mm, rotated rx -180 ry 0 rz 160 deg; joints [-1.46, 69.26, -9.796, -158.726, 61.202, 169.377]
  Set speed (17.8 mm/s)
  Call Extruder(1365.16618)
  MoveL 4175 to (519.05, 439.83, 72) mm, rotated rx -180 ry 0 rz 160 deg; joints [-1.372, 69.616, -10.572, -158.541, 60.828, 169.154]
  Call Extruder(1372.43900)
  MoveL 4176 to (521.22, 440.56, 72) mm, rotated rx 180 ry 0 rz 160 deg; joints [-1.277, 69.965, -11.329, -158.35, 60.466, 168.929]
  Call Extruder(1379.92065)
  MoveL 4177 to (523.42, 441.39, 72) mm, rotated rx -180 ry 0 rz 160 deg; joints [-1.17, 70.323, -12.106, -158.141, 60.098, 168.691]
  Set speed (17.8 mm/s)
  Call Extruder(1387.38862)
  MoveL 4178 to (525.59, 442.3, 72) mm, rotated rx -180 ry 0 rz 160 deg; joints [-1.054, 70.681, -12.878, -157.92, 59.737, 168.446]
  Set speed (17.8 mm/s)
  Call Extruder(1394.77688)
  MoveL 4179 to (527.7, 443.29, 72) mm, rotated rx 180 ry 0 rz 160 deg; joints [-0.932, 71.033, -13.638, -157.69, 59.384, 168.197]
  Set speed (17.8 mm/s)
  Call Extruder(1402.07752)
  MoveL 4180 to (529.74, 444.33, 72) mm, rotated rx -180 ry 0 rz 160 deg; joints [-0.803, 71.38, -14.384, -157.453, 59.043, 167.945]
  Set speed (17.8 mm/s)
  Call Extruder(1409.68263)
  MoveL 4181 to (531.83, 445.5, 72) mm, rotated rx 180 ry 0 rz 160 deg; joints [-0.66, 71.74, -15.155, -157.194, 58.693, 167.675]
  Set speed (17.8 mm/s)
  Call Extruder(1416.84396)
  MoveL 4182 to (533.76, 446.67, 72) mm, rotated rx -180 ry 0 rz 160 deg; joints [-0.519, 72.076, -15.874, -156.941, 58.371, 167.416]
  Set speed (17.8 mm/s)
  Call Extruder(1424.30816)
  MoveL 4183 to (535.72, 447.96, 72) mm, rotated rx 180 ry 0 rz 160 deg; joints [-0.364, 72.424, -16.615, -156.667, 58.043, 167.14]
  Call Extruder(1431.60684)
  MoveL 4184 to (537.59, 449.3, 72) mm, rotated rx -180 ry 0 rz 160 deg; joints [-0.205, 72.76, -17.331, -156.39, 57.731, 166.864]
  Set speed (17.7 mm/s)
  Call Extruder(1439.08845)
  MoveL 4185 to (539.45, 450.73, 72) mm, rotated rx 180 ry 0 rz 160 deg; joints [-0.036, 73.1, -18.054, -156.097, 57.42, 166.577]
  Call Extruder(1446.37935)
  MoveL 4186 to (541.22, 452.2, 72) mm, rotated rx -180 ry 0 rz 160 deg; joints [0.135, 73.428, -18.747, -155.803, 57.125, 166.293]
  Set speed (17.8 mm/s)
  Call Extruder(1453.85235)
  MoveL 4187 to (542.97, 453.77, 72) mm, rotated rx -180 ry 0 rz 160 deg; joints [0.317, 73.758, -19.446, -155.494, 56.833, 165.997]
  Call Extruder(1461.09049)
  MoveL 4188 to (544.61, 455.35, 72) mm, rotated rx 180 ry 0 rz 160 deg; joints [0.5, 74.072, -20.109, -155.186, 56.561, 165.706]
  Set speed (17.8 mm/s)
  Call Extruder(1465.22508)
  MoveL 4189 to (545.52, 456.28, 72) mm, rotated rx 180 ry 0 rz 160 deg; joints [0.606, 74.25, -20.483, -155.008, 56.409, 165.539]
  Set speed (17.8 mm/s)
  Call Extruder(1469.29952)
  MoveL 4190 to (546.4, 457.21, 72) mm, rotated rx 180 ry 0 rz 160 deg; joints [0.713, 74.421, -20.845, -154.83, 56.264, 165.373]
  Set speed (17.8 mm/s)
  Call Extruder(1473.38455)
  MoveL 4191 to (547.26, 458.16, 72) mm, rotated rx -180 ry 0 rz 160 deg; joints [0.822, 74.592, -21.203, -154.65, 56.122, 165.206]
  Call Extruder(1477.48820)
  MoveL 4192 to (548.11, 459.14, 72) mm, rotated rx 180 ry 0 rz 160 deg; joints [0.933, 74.761, -21.558, -154.467, 55.982, 165.038]
  Set speed (17.8 mm/s)
  Call Extruder(1481.59348)
  MoveL 4193 to (548.93, 460.13, 72) mm, rotated rx 180 ry 0 rz 160 deg; joints [1.045, 74.928, -21.908, -154.282, 55.846, 164.869]
  Set speed (17.8 mm/s)
  Call Extruder(1485.74422)
  MoveL 4194 to (549.75, 461.15, 72) mm, rotated rx 180 ry 0 rz 160 deg; joints [1.161, 75.094, -22.256, -154.093, 55.713, 164.697]
  Set speed (17.8 mm/s)
  Call Extruder(1489.78480)
  MoveL 4195 to (550.52, 462.16, 72) mm, rotated rx 180 ry 0 rz 160 deg; joints [1.275, 75.253, -22.59, -153.908, 55.586, 164.529]
  Set speed (17.8 mm/s)
  Call Extruder(1493.44145)
  MoveL 4196 to (551.2, 463.09, 72) mm, rotated rx 180 ry 0 rz 160 deg; joints [1.379, 75.395, -22.886, -153.739, 55.475, 164.377]
  Set speed (17.7 mm/s)
  Call Extruder(1498.02062)
  MoveL 4197 to (552.03, 464.27, 72) mm, rotated rx -180 ry 0 rz 160 deg; joints [1.511, 75.569, -23.25, -153.526, 55.341, 164.187]
  Set speed (17.8 mm/s)
  Call Extruder(1502.09767)
  MoveL 4198 to (552.74, 465.33, 72) mm, rotated rx -180 ry 0 rz 160 deg; joints [1.631, 75.721, -23.568, -153.335, 55.225, 164.017]
  Set speed (17.7 mm/s)
  Call Extruder(1506.32414)
  MoveL 4199 to (553.46, 466.45, 72) mm, rotated rx -180 ry 0 rz 160 deg; joints [1.756, 75.876, -23.891, -153.136, 55.11, 163.842]
  Set speed (17.7 mm/s)
  Call Extruder(1510.36249)
  MoveL 4200 to (554.13, 467.54, 72) mm, rotated rx 180 ry 0 rz 160 deg; joints [1.876, 76.02, -24.192, -152.945, 55.004, 163.674]
  Call Extruder(1514.41940)
  MoveL 4201 to (554.77, 468.63, 72) mm, rotated rx 180 ry 0 rz 160 deg; joints [1.999, 76.163, -24.489, -152.752, 54.902, 163.506]
  Set speed (17.7 mm/s)
  Call Extruder(1519.82464)
  MoveL 4202 to (555.6, 470.12, 72) mm, rotated rx 180 ry 0 rz 160 deg; joints [2.164, 76.347, -24.872, -152.494, 54.772, 163.282]
  Set speed (17.7 mm/s)
  Call Extruder(1522.64533)
  MoveL 4203 to (556.01, 470.9, 72) mm, rotated rx -180 ry 0 rz 160 deg; joints [2.251, 76.441, -25.067, -152.359, 54.707, 163.166]
  Set speed (17.8 mm/s)
  Call Extruder(1526.81072)
  MoveL 4204 to (556.6, 472.07, 72) mm, rotated rx 180 ry 0 rz 160 deg; joints [2.38, 76.576, -25.349, -152.159, 54.615, 162.994]
  Set speed (17.7 mm/s)
  Call Extruder(1532.01696)
  MoveL 4205 to (557.31, 473.55, 72) mm, rotated rx 180 ry 0 rz 160 deg; joints [2.544, 76.741, -25.69, -151.908, 54.507, 162.781]
  Set speed (17.7 mm/s)
  Call Extruder(1535.02080)
  MoveL 4206 to (557.7, 474.41, 72) mm, rotated rx 180 ry 0 rz 160 deg; joints [2.639, 76.832, -25.88, -151.763, 54.449, 162.66]
  Set speed (17.7 mm/s)
  Call Extruder(1539.15353)
  MoveL 4207 to (558.21, 475.6, 72) mm, rotated rx -180 ry 0 rz 160 deg; joints [2.771, 76.954, -26.133, -151.564, 54.373, 162.493]
  Set speed (17.7 mm/s)
  Call Extruder(1543.06003)
  MoveL 4208 to (558.67, 476.74, 72) mm, rotated rx -180 ry 0 rz 160 deg; joints [2.896, 77.068, -26.369, -151.376, 54.304, 162.336]
  Set speed (17.7 mm/s)
  Call Extruder(1547.35681)
  MoveL 4209 to (559.15, 478, 72) mm, rotated rx 180 ry 0 rz 160 deg; joints [3.035, 77.186, -26.614, -151.169, 54.235, 162.165]
  Set speed (17.7 mm/s)
  Call Extruder(1551.46524)
  MoveL 4210 to (559.59, 479.21, 72) mm, rotated rx -180 ry 0 rz 160 deg; joints [3.169, 77.297, -26.844, -150.971, 54.172, 162.003]
  Set speed (17.7 mm/s)
  Call Extruder(1555.60246)
  MoveL 4211 to (560, 480.45, 72) mm, rotated rx -180 ry 0 rz 160 deg; joints [3.304, 77.403, -27.062, -150.772, 54.115, 161.842]
  Set speed (17.7 mm/s)
  Call Extruder(1559.86498)
  MoveL 4212 to (560.41, 481.72, 72) mm, rotated rx 180 ry 0 rz 160 deg; joints [3.444, 77.51, -27.283, -150.567, 54.06, 161.677]
  Set speed (17.7 mm/s)
  Call Extruder(1563.80095)
  MoveL 4213 to (560.75, 482.91, 72) mm, rotated rx -180 ry 0 rz 160 deg; joints [3.575, 77.601, -27.472, -150.379, 54.016, 161.527]
  Set speed (17.7 mm/s)
  Call Extruder(1567.72497)
  MoveL 4214 to (561.08, 484.1, 72) mm, rotated rx 180 ry 0 rz 160 deg; joints [3.706, 77.691, -27.658, -150.191, 53.975, 161.378]
  Call Extruder(0.00000)
  Call Extruder(4.30042)
  MoveL 4215 to (561.4, 485.41, 72) mm, rotated rx -180 ry 0 rz 160 deg; joints [3.85, 77.782, -27.845, -149.987, 53.937, 161.219]
  Call Extruder(8.35200)
  MoveL 4216 to (561.69, 486.65, 72) mm, rotated rx -180 ry 0 rz 160 deg; joints [3.986, 77.866, -28.019, -149.795, 53.904, 161.07]
  Set speed (17.8 mm/s)
  Call Extruder(16.58747)
  MoveL 4217 to (562.19, 489.2, 72) mm, rotated rx 180 ry 0 rz 160 deg; joints [4.266, 78.019, -28.335, -149.407, 53.854, 160.775]
  Set speed (17.7 mm/s)
  Call Extruder(24.73393)
  MoveL 4218 to (562.57, 491.73, 72) mm, rotated rx 180 ry 0 rz 160 deg; joints [4.545, 78.151, -28.607, -149.029, 53.827, 160.494]
  Call Extruder(33.10345)
  MoveL 4219 to (562.86, 494.34, 72) mm, rotated rx -180 ry 0 rz 160 deg; joints [4.833, 78.266, -28.845, -148.647, 53.819, 160.217]
  Set speed (17.8 mm/s)
  Call Extruder(41.21033)
  MoveL 4220 to (563.04, 496.89, 72) mm, rotated rx 180 ry 0 rz 160 deg; joints [5.114, 78.358, -29.033, -148.283, 53.832, 159.962]
  Set speed (17.8 mm/s)
  Call Extruder(49.41542)
  MoveL 4221 to (563.11, 499.47, 72) mm, rotated rx 180 ry 0 rz 160 deg; joints [5.399, 78.429, -29.18, -147.922, 53.866, 159.716]
  Set speed (17.8 mm/s)
  Call Extruder(57.51128)
  MoveL 4222 to (563.08, 502.02, 72) mm, rotated rx -180 ry 0 rz 160 deg; joints [5.682, 78.479, -29.282, -147.574, 53.92, 159.488]
  Set speed (17.8 mm/s)
  Call Extruder(65.82577)
  MoveL 4223 to (562.95, 504.63, 72) mm, rotated rx -180 ry 0 rz 160 deg; joints [5.972, 78.51, -29.345, -147.224, 53.995, 159.269]
  Set speed (17.8 mm/s)
  Call Extruder(73.95087)
  MoveL 4224 to (562.71, 507.18, 72) mm, rotated rx 180 ry 0 rz 160 deg; joints [6.257, 78.517, -29.36, -146.893, 54.09, 159.071]
  Set speed (17.8 mm/s)
  Call Extruder(82.32533)
  MoveL 4225 to (562.35, 509.79, 72) mm, rotated rx 180 ry 0 rz 160 deg; joints [6.55, 78.503, -29.331, -146.561, 54.208, 158.883]
  Set speed (17.8 mm/s)
  Call Extruder(90.42373)
  MoveL 4226 to (561.91, 512.3, 72) mm, rotated rx 180 ry 0 rz 160 deg; joints [6.833, 78.468, -29.259, -146.251, 54.341, 158.719]
  Set speed (17.8 mm/s)
  Call Extruder(98.69358)
  MoveL 4227 to (561.35, 514.84, 72) mm, rotated rx -180 ry 0 rz 160 deg; joints [7.121, 78.411, -29.141, -145.945, 54.496, 158.568]
  Set speed (17.7 mm/s)
  Call Extruder(102.77552)
  MoveL 4228 to (561.03, 516.08, 72) mm, rotated rx 180 ry 0 rz 160 deg; joints [7.263, 78.373, -29.065, -145.798, 54.581, 158.501]
  Set speed (17.7 mm/s)
  Call Extruder(106.99374)
  MoveL 4229 to (560.68, 517.36, 72) mm, rotated rx -180 ry 0 rz 160 deg; joints [7.41, 78.332, -28.98, -145.649, 54.67, 158.434]
  Set speed (17.7 mm/s)
  Call Extruder(111.03015)
  MoveL 4230 to (560.32, 518.58, 72) mm, rotated rx 180 ry 0 rz 160 deg; joints [7.549, 78.285, -28.883, -145.51, 54.763, 158.377]
  Set speed (17.7 mm/s)
  Call Extruder(114.96931)
  MoveL 4231 to (559.94, 519.76, 72) mm, rotated rx 180 ry 0 rz 160 deg; joints [7.685, 78.236, -28.783, -145.376, 54.855, 158.324]
  Set speed (17.8 mm/s)
  Call Extruder(123.29260)
  MoveL 4232 to (559.07, 522.23, 72) mm, rotated rx -180 ry 0 rz 160 deg; joints [7.971, 78.116, -28.535, -145.102, 55.066, 158.226]
  Set speed (17.7 mm/s)
  Call Extruder(127.38783)
  MoveL 4233 to (558.6, 523.43, 72) mm, rotated rx 180 ry 0 rz 160 deg; joints [8.111, 78.048, -28.395, -144.973, 55.177, 158.186]
  Set speed (17.7 mm/s)
  Call Extruder(131.35896)
  MoveL 4234 to (558.13, 524.58, 72) mm, rotated rx -180 ry 0 rz 160 deg; joints [8.247, 77.98, -28.255, -144.848, 55.287, 158.149]
  Call Extruder(135.61569)
  MoveL 4235 to (557.59, 525.81, 72) mm, rotated rx 180 ry 0 rz 160 deg; joints [8.391, 77.899, -28.087, -144.72, 55.411, 158.117]
  Set speed (17.7 mm/s)
  Call Extruder(139.55201)
  MoveL 4236 to (557.08, 526.93, 72) mm, rotated rx -180 ry 0 rz 160 deg; joints [8.524, 77.822, -27.929, -144.603, 55.527, 158.09]
  Set speed (17.7 mm/s)
  Call Extruder(142.73886)
  MoveL 4237 to (556.65, 527.84, 72) mm, rotated rx 180 ry 0 rz 160 deg; joints [8.631, 77.757, -27.794, -144.51, 55.624, 158.07]
  Set speed (17.8 mm/s)
  Call Extruder(149.97415)
  MoveL 4238 to (555.61, 529.86, 72) mm, rotated rx 180 ry 0 rz 160 deg; joints [8.873, 77.596, -27.463, -144.306, 55.853, 158.038]
  Set speed (17.8 mm/s)
  Call Extruder(156.05598)
  MoveL 4239 to (554.67, 531.54, 72) mm, rotated rx 180 ry 0 rz 160 deg; joints [9.075, 77.449, -27.158, -144.142, 56.056, 158.023]
  Set speed (17.7 mm/s)
  Call Extruder(160.97281)
  MoveL 4240 to (553.89, 532.87, 72) mm, rotated rx -180 ry 0 rz 160 deg; joints [9.236, 77.324, -26.9, -144.014, 56.224, 158.016]
  Set speed (17.8 mm/s)
  Call Extruder(164.24113)
  MoveL 4241 to (553.34, 533.74, 72) mm, rotated rx -180 ry 0 rz 160 deg; joints [9.343, 77.237, -26.72, -143.932, 56.34, 158.016]
  Call Extruder(167.77998)
  MoveL 4242 to (552.74, 534.67, 72) mm, rotated rx -180 ry 0 rz 160 deg; joints [9.458, 77.141, -26.52, -143.844, 56.467, 158.018]
  Set speed (17.7 mm/s)
  Call Extruder(172.50609)
  MoveL 4243 to (551.91, 535.91, 72) mm, rotated rx 180 ry 0 rz 160 deg; joints [9.61, 77.006, -26.242, -143.731, 56.64, 158.027]
  Set speed (17.8 mm/s)
  Call Extruder(176.68762)
  MoveL 4244 to (551.15, 536.98, 72) mm, rotated rx 180 ry 0 rz 160 deg; joints [9.744, 76.884, -25.988, -143.634, 56.796, 158.038]
  Set speed (17.8 mm/s)
  Call Extruder(180.74204)
  MoveL 4245 to (550.39, 538.01, 72) mm, rotated rx 180 ry 0 rz 160 deg; joints [9.873, 76.761, -25.732, -143.543, 56.95, 158.054]
  Set speed (17.8 mm/s)
  Call Extruder(184.76509)
  MoveL 4246 to (549.62, 539.01, 72) mm, rotated rx -180 ry 0 rz 160 deg; joints [10, 76.635, -25.471, -143.455, 57.106, 158.074]
  Call Extruder(188.86100)
  MoveL 4247 to (548.81, 540.01, 72) mm, rotated rx -180 ry 0 rz 160 deg; joints [10.128, 76.504, -25.198, -143.368, 57.268, 158.098]
  Call Extruder(193.05546)
  MoveL 4248 to (547.97, 541.02, 72) mm, rotated rx 180 ry 0 rz 160 deg; joints [10.257, 76.365, -24.909, -143.282, 57.436, 158.127]
  Set speed (17.8 mm/s)
  Call Extruder(197.10178)
  MoveL 4249 to (547.13, 541.99, 72) mm, rotated rx -180 ry 0 rz 160 deg; joints [10.381, 76.228, -24.625, -143.202, 57.601, 158.159]
  Set speed (17.7 mm/s)
  Call Extruder(203.44830)
  MoveL 4250 to (545.78, 543.45, 72) mm, rotated rx -180 ry 0 rz 160 deg; joints [10.573, 76.007, -24.164, -143.082, 57.864, 158.216]
  Call Extruder(209.49457)
  MoveL 4251 to (544.45, 544.81, 72) mm, rotated rx 180 ry 0 rz 160 deg; joints [10.753, 75.789, -23.709, -142.974, 58.12, 158.28]
  Set speed (17.8 mm/s)
  Call Extruder(213.49681)
  MoveL 4252 to (543.55, 545.69, 72) mm, rotated rx 180 ry 0 rz 160 deg; joints [10.871, 75.641, -23.4, -142.905, 58.292, 158.326]
  Set speed (17.8 mm/s)
  Call Extruder(217.59416)
  MoveL 4253 to (542.61, 546.57, 72) mm, rotated rx 180 ry 0 rz 160 deg; joints [10.99, 75.486, -23.077, -142.838, 58.47, 158.377]
  Set speed (17.8 mm/s)
  Call Extruder(221.75978)
  MoveL 4254 to (541.63, 547.44, 72) mm, rotated rx -180 ry 0 rz 160 deg; joints [11.11, 75.326, -22.742, -142.772, 58.654, 158.433]
  Set speed (17.8 mm/s)
  Call Extruder(225.92504)
  MoveL 4255 to (540.63, 548.3, 72) mm, rotated rx -180 ry 0 rz 160 deg; joints [11.228, 75.163, -22.401, -142.709, 58.839, 158.492]
  Set speed (17.8 mm/s)
  Call Extruder(229.93481)
  MoveL 4256 to (539.66, 549.1, 72) mm, rotated rx -180 ry 0 rz 160 deg; joints [11.34, 75.003, -22.067, -142.651, 59.019, 158.553]
  Set speed (17.8 mm/s)
  Call Extruder(234.03478)
  MoveL 4257 to (538.65, 549.9, 72) mm, rotated rx 180 ry 0 rz 160 deg; joints [11.453, 74.838, -21.72, -142.594, 59.204, 158.618]
  Call Extruder(238.12821)
  MoveL 4258 to (537.62, 550.68, 72) mm, rotated rx 180 ry 0 rz 160 deg; joints [11.565, 74.671, -21.368, -142.54, 59.391, 158.687]
  Set speed (17.8 mm/s)
  Call Extruder(242.27120)
  MoveL 4259 to (536.57, 551.45, 72) mm, rotated rx 180 ry 0 rz 160 deg; joints [11.676, 74.499, -21.007, -142.488, 59.582, 158.76]
  Set speed (17.8 mm/s)
  Call Extruder(246.30604)
  MoveL 4260 to (535.52, 552.17, 72) mm, rotated rx 180 ry 0 rz 160 deg; joints [11.783, 74.329, -20.65, -142.439, 59.769, 158.834]
  Set speed (17.8 mm/s)
  Call Extruder(250.47386)
  MoveL 4261 to (534.43, 552.9, 72) mm, rotated rx -180 ry 0 rz 160 deg; joints [11.891, 74.152, -20.276, -142.392, 59.963, 158.914]
  Set speed (17.7 mm/s)
  Call Extruder(254.52770)
  MoveL 4262 to (533.36, 553.58, 72) mm, rotated rx -180 ry 0 rz 160 deg; joints [11.994, 73.977, -19.909, -142.348, 60.153, 158.994]
  Set speed (17.8 mm/s)
  Call Extruder(258.82166)
  MoveL 4263 to (532.2, 554.28, 72) mm, rotated rx 180 ry 0 rz 160 deg; joints [12.102, 73.791, -19.515, -142.305, 60.356, 159.082]
  Set speed (17.8 mm/s)
  Call Extruder(262.74353)
  MoveL 4264 to (531.14, 554.9, 72) mm, rotated rx 180 ry 0 rz 160 deg; joints [12.199, 73.618, -19.151, -142.267, 60.542, 159.166]
  Set speed (17.8 mm/s)
  Call Extruder(266.26845)
  MoveL 4265 to (530.17, 555.44, 72) mm, rotated rx -180 ry 0 rz 160 deg; joints [12.284, 73.462, -18.82, -142.236, 60.71, 159.244]
  Set speed (17.7 mm/s)
  Call Extruder(272.09000)
  MoveL 4266 to (528.55, 556.3, 72) mm, rotated rx 180 ry 0 rz 160 deg; joints [12.423, 73.202, -18.27, -142.187, 60.989, 159.375]
  Set speed (17.8 mm/s)
  Call Extruder(279.07542)
  MoveL 4267 to (526.57, 557.25, 72) mm, rotated rx 180 ry 0 rz 160 deg; joints [12.582, 72.885, -17.597, -142.137, 61.326, 159.542]
  Set speed (17.7 mm/s)
  Call Extruder(283.33188)
  MoveL 4268 to (525.35, 557.8, 72) mm, rotated rx 180 ry 0 rz 160 deg; joints [12.676, 72.69, -17.182, -142.11, 61.532, 159.648]
  Set speed (17.7 mm/s)
  Call Extruder(287.34765)
  MoveL 4269 to (524.19, 558.3, 72) mm, rotated rx 180 ry 0 rz 160 deg; joints [12.764, 72.506, -16.79, -142.085, 61.726, 159.749]
  Set speed (17.7 mm/s)
  Call Extruder(291.55550)
  MoveL 4270 to (522.96, 558.79, 72) mm, rotated rx 180 ry 0 rz 160 deg; joints [12.852, 72.31, -16.374, -142.064, 61.931, 159.858]
  Call Extruder(295.80445)
  MoveL 4271 to (521.71, 559.27, 72) mm, rotated rx -180 ry 0 rz 160 deg; joints [12.941, 72.114, -15.954, -142.043, 62.138, 159.97]
  Set speed (17.8 mm/s)
  Call Extruder(303.76359)
  MoveL 4272 to (519.35, 560.08, 72) mm, rotated rx -180 ry 0 rz 160 deg; joints [13.098, 71.74, -15.155, -142.013, 62.526, 160.187]
  Set speed (17.7 mm/s)
  Call Extruder(307.97303)
  MoveL 4273 to (518.08, 560.47, 72) mm, rotated rx 180 ry 0 rz 160 deg; joints [13.177, 71.541, -14.729, -142.001, 62.732, 160.306]
  Call Extruder(311.93403)
  MoveL 4274 to (516.89, 560.82, 72) mm, rotated rx 180 ry 0 rz 160 deg; joints [13.251, 71.354, -14.328, -141.991, 62.925, 160.419]
  Set speed (17.7 mm/s)
  Call Extruder(315.64491)
  MoveL 4275 to (515.76, 561.11, 72) mm, rotated rx -180 ry 0 rz 160 deg; joints [13.316, 71.178, -13.949, -141.985, 63.107, 160.527]
  Call Extruder(320.23122)
  MoveL 4276 to (514.36, 561.46, 72) mm, rotated rx 180 ry 0 rz 160 deg; joints [13.396, 70.96, -13.481, -141.979, 63.331, 160.662]
  Set speed (17.8 mm/s)
  Call Extruder(328.51560)
  MoveL 4277 to (511.81, 562, 72) mm, rotated rx 180 ry 0 rz 160 deg; joints [13.531, 70.565, -12.628, -141.977, 63.735, 160.913]
  Set speed (17.7 mm/s)
  Call Extruder(336.78723)
  MoveL 4278 to (509.25, 562.44, 72) mm, rotated rx -180 ry 0 rz 160 deg; joints [13.655, 70.169, -11.772, -141.985, 64.138, 161.172]
  Call Extruder(344.90640)
  MoveL 4279 to (506.71, 562.76, 72) mm, rotated rx 180 ry 0 rz 160 deg; joints [13.766, 69.78, -10.929, -142.003, 64.532, 161.432]
  Set speed (17.8 mm/s)
  Call Extruder(353.15143)
  MoveL 4280 to (504.13, 562.98, 72) mm, rotated rx 180 ry 0 rz 160 deg; joints [13.868, 69.385, -10.07, -142.03, 64.93, 161.702]
  Set speed (17.8 mm/s)
  Call Extruder(361.41385)
  MoveL 4281 to (501.53, 563.1, 72) mm, rotated rx 180 ry 0 rz 160 deg; joints [13.959, 68.991, -9.208, -142.069, 65.326, 161.978]
  Set speed (17.8 mm/s)
  Call Extruder(369.53940)
  MoveL 4282 to (498.98, 563.11, 72) mm, rotated rx 180 ry 0 rz 160 deg; joints [14.037, 68.604, -8.362, -142.116, 65.713, 162.255]
  Set speed (10.0 mm/s)
  MoveL 4283 to (498.98, 563.11, 76) mm, rotated rx -180 ry 0 rz 160 deg; joints [14.037, 67.938, -7.989, -142.034, 65.482, 162.057]
  Set speed (120.0 mm/s)
  MoveL 4284 to (499, 563.75, 76) mm, rotated rx 180 ry 0 rz 160 deg; joints [14.113, 67.965, -8.048, -141.945, 65.48, 162.002]
  Set speed (17.8 mm/s)
  Call Extruder(377.95724)
  MoveL 4285 to (496.34, 563.65, 76) mm, rotated rx 180 ry 0 rz 160 deg; joints [14.182, 67.564, -7.172, -142.006, 65.875, 162.293]
  Set speed (17.8 mm/s)
  Call Extruder(386.25646)
  MoveL 4286 to (493.73, 563.45, 76) mm, rotated rx 180 ry 0 rz 160 deg; joints [14.237, 67.172, -6.313, -142.075, 66.26, 162.584]
  Set speed (17.8 mm/s)
  Call Extruder(394.45732)
  MoveL 4287 to (491.17, 563.14, 76) mm, rotated rx 180 ry 0 rz 160 deg; joints [14.279, 66.787, -5.468, -142.155, 66.637, 162.876]
  Set speed (17.8 mm/s)
  Call Extruder(402.70742)
  MoveL 4288 to (488.6, 562.73, 76) mm, rotated rx -180 ry 0 rz 160 deg; joints [14.309, 66.404, -4.622, -142.246, 67.01, 163.172]
  Call Extruder(411.10868)
  MoveL 4289 to (486.01, 562.2, 76) mm, rotated rx 180 ry 0 rz 160 deg; joints [14.325, 66.018, -3.768, -142.349, 67.386, 163.476]
  Set speed (17.8 mm/s)
  Call Extruder(415.21211)
  MoveL 4290 to (484.75, 561.9, 76) mm, rotated rx 180 ry 0 rz 160 deg; joints [14.328, 65.832, -3.354, -142.404, 67.566, 163.625]
  Set speed (17.8 mm/s)
  Call Extruder(419.24684)
  MoveL 4291 to (483.52, 561.59, 76) mm, rotated rx -180 ry 0 rz 160 deg; joints [14.328, 65.65, -2.95, -142.459, 67.743, 163.772]
  Call Extruder(423.42400)
  MoveL 4292 to (482.26, 561.23, 76) mm, rotated rx 180 ry 0 rz 160 deg; joints [14.324, 65.463, -2.533, -142.52, 67.924, 163.924]
  Set speed (17.8 mm/s)
  Call Extruder(427.69743)
  MoveL 4293 to (480.97, 560.85, 76) mm, rotated rx 180 ry 0 rz 160 deg; joints [14.317, 65.273, -2.108, -142.584, 68.108, 164.08]
  Set speed (17.8 mm/s)
  Call Extruder(435.79769)
  MoveL 4294 to (478.55, 560.04, 76) mm, rotated rx -180 ry 0 rz 160 deg; joints [14.293, 64.916, -1.311, -142.716, 68.452, 164.378]
  Set speed (17.8 mm/s)
  Call Extruder(440.05158)
  MoveL 4295 to (477.29, 559.57, 76) mm, rotated rx 180 ry 0 rz 160 deg; joints [14.274, 64.731, -0.896, -142.791, 68.63, 164.534]
  Call Extruder(444.06929)
  MoveL 4296 to (476.11, 559.11, 76) mm, rotated rx -180 ry 0 rz 160 deg; joints [14.254, 64.558, -0.507, -142.862, 68.797, 164.682]
  Set speed (17.8 mm/s)
  Call Extruder(451.42519)
  MoveL 4297 to (473.98, 558.21, 76) mm, rotated rx 180 ry 0 rz 160 deg; joints [14.208, 64.246, 0.197, -143.001, 69.098, 164.952]
  Set speed (17.8 mm/s)
  Call Extruder(456.49446)
  MoveL 4298 to (472.53, 557.54, 76) mm, rotated rx -180 ry 0 rz 160 deg; joints [14.169, 64.033, 0.677, -143.102, 69.301, 165.138]
  Set speed (17.8 mm/s)
  Call Extruder(460.68569)
  MoveL 4299 to (471.34, 556.95, 76) mm, rotated rx 180 ry 0 rz 160 deg; joints [14.133, 63.86, 1.07, -143.189, 69.468, 165.292]
  Set speed (17.8 mm/s)
  Call Extruder(463.70635)
  MoveL 4300 to (470.5, 556.52, 76) mm, rotated rx 180 ry 0 rz 160 deg; joints [14.105, 63.736, 1.351, -143.253, 69.587, 165.403]
  Set speed (17.8 mm/s)
  Call Extruder(469.10097)
  MoveL 4301 to (469, 555.72, 76) mm, rotated rx 180 ry 0 rz 160 deg; joints [14.049, 63.517, 1.848, -143.372, 69.796, 165.6]
  Set speed (17.8 mm/s)
  Call Extruder(473.02720)
  MoveL 4302 to (467.93, 555.1, 76) mm, rotated rx 180 ry 0 rz 160 deg; joints [14.005, 63.36, 2.206, -143.462, 69.946, 165.743]
  Set speed (17.8 mm/s)
  Call Extruder(477.25142)
  MoveL 4303 to (466.78, 554.42, 76) mm, rotated rx 180 ry 0 rz 160 deg; joints [13.953, 63.193, 2.588, -143.561, 70.106, 165.897]
  Set speed (17.8 mm/s)
  Call Extruder(481.39324)
  MoveL 4304 to (465.67, 553.73, 76) mm, rotated rx 180 ry 0 rz 160 deg; joints [13.899, 63.031, 2.957, -143.662, 70.26, 166.047]
  Set speed (17.8 mm/s)
  Call Extruder(485.42989)
  MoveL 4305 to (464.61, 553.03, 76) mm, rotated rx 180 ry 0 rz 160 deg; joints [13.842, 62.875, 3.313, -143.762, 70.408, 166.193]
  Set speed (17.8 mm/s)
  Call Extruder(489.62412)
  MoveL 4306 to (463.52, 552.28, 76) mm, rotated rx 180 ry 0 rz 160 deg; joints [13.78, 62.716, 3.68, -143.87, 70.56, 166.344]
  Set speed (17.8 mm/s)
  Call Extruder(493.73449)
  MoveL 4307 to (462.46, 551.53, 76) mm, rotated rx 180 ry 0 rz 160 deg; joints [13.716, 62.562, 4.034, -143.978, 70.707, 166.491]
  Set speed (17.8 mm/s)
  Call Extruder(497.91849)
  MoveL 4308 to (461.4, 550.75, 76) mm, rotated rx -180 ry 0 rz 160 deg; joints [13.646, 62.407, 4.39, -144.091, 70.853, 166.64]
  Call Extruder(502.09415)
  MoveL 4309 to (460.36, 549.94, 76) mm, rotated rx -180 ry 0 rz 160 deg; joints [13.572, 62.255, 4.741, -144.207, 70.998, 166.787]
  Set speed (17.8 mm/s)
  Call Extruder(506.17456)
  MoveL 4310 to (459.37, 549.13, 76) mm, rotated rx 180 ry 0 rz 160 deg; joints [13.497, 62.109, 5.078, -144.323, 71.136, 166.931]
  Set speed (17.8 mm/s)
  Call Extruder(510.36962)
  MoveL 4311 to (458.35, 548.28, 76) mm, rotated rx 180 ry 0 rz 160 deg; joints [13.416, 61.961, 5.421, -144.445, 71.276, 167.078]
  Set speed (17.8 mm/s)
  Call Extruder(513.89856)
  MoveL 4312 to (457.52, 547.54, 76) mm, rotated rx 180 ry 0 rz 160 deg; joints [13.345, 61.838, 5.706, -144.55, 71.392, 167.2]
  Set speed (17.8 mm/s)
  Call Extruder(519.15008)
  MoveL 4313 to (456.3, 546.42, 76) mm, rotated rx -180 ry 0 rz 160 deg; joints [13.234, 61.66, 6.121, -144.71, 71.56, 167.381]
  Set speed (17.8 mm/s)
  Call Extruder(522.35706)
  MoveL 4314 to (455.57, 545.73, 76) mm, rotated rx -180 ry 0 rz 160 deg; joints [13.163, 61.553, 6.37, -144.81, 71.661, 167.491]
  Set speed (17.8 mm/s)
  Call Extruder(526.85922)
  MoveL 4315 to (454.56, 544.73, 76) mm, rotated rx -180 ry 0 rz 160 deg; joints [13.06, 61.405, 6.715, -144.953, 71.801, 167.643]
  Set speed (17.8 mm/s)
  Call Extruder(530.96405)
  MoveL 4316 to (453.67, 543.79, 76) mm, rotated rx -180 ry 0 rz 160 deg; joints [12.963, 61.273, 7.024, -145.087, 71.925, 167.781]
  Set speed (17.8 mm/s)
  Call Extruder(535.11058)
  MoveL 4317 to (452.78, 542.84, 76) mm, rotated rx 180 ry 0 rz 160 deg; joints [12.861, 61.142, 7.331, -145.224, 72.048, 167.919]
  Set speed (17.8 mm/s)
  Call Extruder(538.43004)
  MoveL 4318 to (452.08, 542.05, 76) mm, rotated rx -180 ry 0 rz 160 deg; joints [12.776, 61.039, 7.573, -145.336, 72.144, 168.029]
  Set speed (17.8 mm/s)
  Call Extruder(543.57920)
  MoveL 4319 to (451.02, 540.82, 76) mm, rotated rx -180 ry 0 rz 160 deg; joints [12.641, 60.882, 7.94, -145.514, 72.29, 168.197]
  Set speed (17.8 mm/s)
  Call Extruder(547.54826)
  MoveL 4320 to (450.24, 539.85, 76) mm, rotated rx -180 ry 0 rz 160 deg; joints [12.533, 60.765, 8.217, -145.654, 72.399, 168.325]
  Call Extruder(551.70614)
  MoveL 4321 to (449.43, 538.82, 76) mm, rotated rx 180 ry 0 rz 160 deg; joints [12.416, 60.644, 8.501, -145.803, 72.511, 168.458]
  Set speed (17.8 mm/s)
  Call Extruder(555.84028)
  MoveL 4322 to (448.64, 537.78, 76) mm, rotated rx 180 ry 0 rz 160 deg; joints [12.297, 60.527, 8.777, -145.953, 72.619, 168.588]
  Set speed (17.8 mm/s)
  Call Extruder(559.90969)
  MoveL 4323 to (447.9, 536.74, 76) mm, rotated rx 180 ry 0 rz 160 deg; joints [12.176, 60.415, 9.043, -146.104, 72.723, 168.715]
  Set speed (17.8 mm/s)
  Call Extruder(564.07780)
  MoveL 4324 to (447.15, 535.66, 76) mm, rotated rx 180 ry 0 rz 160 deg; joints [12.049, 60.303, 9.31, -146.261, 72.826, 168.844]
  Call Extruder(568.25415)
  MoveL 4325 to (446.42, 534.56, 76) mm, rotated rx 180 ry 0 rz 160 deg; joints [11.918, 60.193, 9.57, -146.421, 72.926, 168.971]
  Set speed (17.8 mm/s)
  Call Extruder(572.37880)
  MoveL 4326 to (445.73, 533.46, 76) mm, rotated rx -180 ry 0 rz 160 deg; joints [11.786, 60.088, 9.82, -146.582, 73.022, 169.094]
  Set speed (17.8 mm/s)
  Call Extruder(576.46077)
  MoveL 4327 to (445.07, 532.36, 76) mm, rotated rx 180 ry 0 rz 160 deg; joints [11.651, 59.986, 10.062, -146.743, 73.114, 169.215]
  Set speed (17.8 mm/s)
  Call Extruder(580.65733)
  MoveL 4328 to (444.41, 531.21, 76) mm, rotated rx -180 ry 0 rz 160 deg; joints [11.51, 59.885, 10.304, -146.911, 73.205, 169.337]
  Call Extruder(584.71852)
  MoveL 4329 to (443.79, 530.09, 76) mm, rotated rx 180 ry 0 rz 160 deg; joints [11.37, 59.79, 10.53, -147.076, 73.29, 169.454]
  Call Extruder(588.91978)
  MoveL 4330 to (443.18, 528.92, 76) mm, rotated rx -180 ry 0 rz 160 deg; joints [11.223, 59.695, 10.759, -147.249, 73.375, 169.572]
  Set speed (17.8 mm/s)
  Call Extruder(592.99765)
  MoveL 4331 to (442.61, 527.77, 76) mm, rotated rx 180 ry 0 rz 160 deg; joints [11.077, 59.605, 10.973, -147.419, 73.454, 169.685]
  Set speed (17.8 mm/s)
  Call Extruder(597.27610)
  MoveL 4332 to (442.04, 526.54, 76) mm, rotated rx -180 ry 0 rz 160 deg; joints [10.92, 59.515, 11.189, -147.6, 73.532, 169.802]
  Call Extruder(601.24623)
  MoveL 4333 to (441.52, 525.4, 76) mm, rotated rx 180 ry 0 rz 160 deg; joints [10.773, 59.434, 11.386, -147.769, 73.603, 169.908]
  Set speed (17.8 mm/s)
  Call Extruder(605.56966)
  MoveL 4334 to (441, 524.15, 76) mm, rotated rx -180 ry 0 rz 160 deg; joints [10.609, 59.35, 11.589, -147.956, 73.675, 170.022]
  Set speed (17.8 mm/s)
  Call Extruder(609.56911)
  MoveL 4335 to (440.53, 522.98, 76) mm, rotated rx 180 ry 0 rz 160 deg; joints [10.456, 59.273, 11.773, -148.13, 73.74, 170.125]
  Set speed (17.8 mm/s)
  Call Extruder(613.83079)
  MoveL 4336 to (440.07, 521.72, 76) mm, rotated rx 180 ry 0 rz 160 deg; joints [10.289, 59.196, 11.958, -148.318, 73.804, 170.232]
  Set speed (17.8 mm/s)
  Call Extruder(617.85486)
  MoveL 4337 to (439.64, 520.53, 76) mm, rotated rx 180 ry 0 rz 160 deg; joints [10.13, 59.126, 12.129, -148.496, 73.862, 170.332]
  Set speed (17.8 mm/s)
  Call Extruder(622.13792)
  MoveL 4338 to (439.23, 519.25, 76) mm, rotated rx -180 ry 0 rz 160 deg; joints [9.957, 59.055, 12.299, -148.689, 73.919, 170.436]
  Set speed (17.8 mm/s)
  Call Extruder(626.29331)
  MoveL 4339 to (438.84, 518, 76) mm, rotated rx -180 ry 0 rz 160 deg; joints [9.788, 58.989, 12.46, -148.876, 73.972, 170.535]
  Set speed (17.8 mm/s)
  Call Extruder(630.42660)
  MoveL 4340 to (438.49, 516.75, 76) mm, rotated rx -180 ry 0 rz 160 deg; joints [9.617, 58.927, 12.61, -149.065, 74.019, 170.631]
  Set speed (17.8 mm/s)
  Call Extruder(634.52565)
  MoveL 4341 to (438.16, 515.5, 76) mm, rotated rx 180 ry 0 rz 160 deg; joints [9.446, 58.868, 12.754, -149.253, 74.064, 170.724]
  Set speed (17.8 mm/s)
  Call Extruder(638.10366)
  MoveL 4342 to (437.9, 514.4, 76) mm, rotated rx -180 ry 0 rz 160 deg; joints [9.294, 58.82, 12.87, -149.419, 74.099, 170.803]
  Set speed (17.7 mm/s)
  Call Extruder(643.55558)
  MoveL 4343 to (437.53, 512.73, 76) mm, rotated rx 180 ry 0 rz 160 deg; joints [9.061, 58.751, 13.039, -149.672, 74.148, 170.921]
  Set speed (17.8 mm/s)
  Call Extruder(651.16955)
  MoveL 4344 to (437.09, 510.37, 76) mm, rotated rx 180 ry 0 rz 160 deg; joints [8.73, 58.663, 13.252, -150.03, 74.204, 171.079]
  Set speed (17.8 mm/s)
  Call Extruder(659.44307)
  MoveL 4345 to (436.72, 507.79, 76) mm, rotated rx 180 ry 0 rz 160 deg; joints [8.364, 58.581, 13.453, -150.423, 74.251, 171.243]
  Set speed (17.8 mm/s)
  Call Extruder(667.71724)
  MoveL 4346 to (436.46, 505.2, 76) mm, rotated rx 180 ry 0 rz 160 deg; joints [7.992, 58.512, 13.621, -150.819, 74.282, 171.397]
  Set speed (17.8 mm/s)
  Call Extruder(675.83924)
  MoveL 4347 to (436.3, 502.64, 76) mm, rotated rx 180 ry 0 rz 160 deg; joints [7.622, 58.457, 13.756, -151.209, 74.296, 171.54]
  Set speed (17.8 mm/s)
  Call Extruder(684.18524)
  MoveL 4348 to (436.24, 500.01, 76) mm, rotated rx 180 ry 0 rz 160 deg; joints [7.239, 58.414, 13.861, -151.611, 74.295, 171.677]
  Set speed (17.8 mm/s)
  Call Extruder(691.71564)
  MoveL 4349 to (436.29, 497.64, 76) mm, rotated rx -180 ry 0 rz 160 deg; joints [6.891, 58.387, 13.926, -151.974, 74.279, 171.793]
  Set speed (17.8 mm/s)
  Call Extruder(699.08564)
  MoveL 4350 to (436.42, 495.32, 76) mm, rotated rx 180 ry 0 rz 160 deg; joints [6.549, 58.372, 13.965, -152.329, 74.251, 171.9]
  Call Extruder(706.45348)
  MoveL 4351 to (436.63, 493.01, 76) mm, rotated rx 180 ry 0 rz 160 deg; joints [6.206, 58.367, 13.977, -152.682, 74.209, 171.999]
  Call Extruder(713.89621)
  MoveL 4352 to (436.93, 490.68, 76) mm, rotated rx 180 ry 0 rz 160 deg; joints [5.86, 58.373, 13.962, -153.037, 74.153, 172.092]
  Set speed (17.8 mm/s)
  Call Extruder(721.25117)
  MoveL 4353 to (437.31, 488.4, 76) mm, rotated rx -180 ry 0 rz 160 deg; joints [5.519, 58.389, 13.922, -153.386, 74.086, 172.177]
  Set speed (17.8 mm/s)
  Call Extruder(728.80786)
  MoveL 4354 to (437.79, 486.06, 76) mm, rotated rx 180 ry 0 rz 160 deg; joints [5.17, 58.417, 13.854, -153.741, 74.002, 172.257]
  Call Extruder(736.30755)
  MoveL 4355 to (438.35, 483.77, 76) mm, rotated rx 180 ry 0 rz 160 deg; joints [4.825, 58.456, 13.759, -154.089, 73.905, 172.329]
  Set speed (17.8 mm/s)
  Call Extruder(743.75680)
  MoveL 4356 to (438.99, 481.51, 76) mm, rotated rx 180 ry 0 rz 160 deg; joints [4.486, 58.505, 13.638, -154.43, 73.796, 172.394]
  Set speed (17.8 mm/s)
  Call Extruder(751.20708)
  MoveL 4357 to (439.71, 479.27, 76) mm, rotated rx 180 ry 0 rz 160 deg; joints [4.151, 58.566, 13.49, -154.765, 73.673, 172.453]
  Set speed (17.8 mm/s)
  Call Extruder(758.64305)
  MoveL 4358 to (440.51, 477.07, 76) mm, rotated rx 180 ry 0 rz 160 deg; joints [3.82, 58.637, 13.317, -155.094, 73.537, 172.504]
  Set speed (17.8 mm/s)
  Call Extruder(765.29494)
  MoveL 4359 to (441.3, 475.13, 76) mm, rotated rx 180 ry 0 rz 160 deg; joints [3.528, 58.709, 13.141, -155.383, 73.405, 172.544]
  Set speed (17.8 mm/s)
  Call Extruder(773.48413)
  MoveL 4360 to (442.35, 472.77, 76) mm, rotated rx -180 ry 0 rz 160 deg; joints [3.176, 58.81, 12.896, -155.73, 73.227, 172.587]
  Set speed (17.8 mm/s)
  Call Extruder(781.08520)
  MoveL 4361 to (443.41, 470.63, 76) mm, rotated rx -180 ry 0 rz 160 deg; joints [2.855, 58.915, 12.64, -156.044, 73.049, 172.619]
  Call Extruder(788.38391)
  MoveL 4362 to (444.51, 468.61, 76) mm, rotated rx 180 ry 0 rz 160 deg; joints [2.554, 59.026, 12.37, -156.337, 72.865, 172.644]
  Set speed (17.8 mm/s)
  Call Extruder(795.98213)
  MoveL 4363 to (445.73, 466.54, 76) mm, rotated rx -180 ry 0 rz 160 deg; joints [2.247, 59.152, 12.065, -156.633, 72.662, 172.663]
  Set speed (17.8 mm/s)
  Call Extruder(803.34528)
  MoveL 4364 to (446.98, 464.59, 76) mm, rotated rx 180 ry 0 rz 160 deg; joints [1.958, 59.285, 11.745, -156.91, 72.452, 172.676]
  Set speed (17.8 mm/s)
  Call Extruder(810.79165)
  MoveL 4365 to (448.32, 462.66, 76) mm, rotated rx -180 ry 0 rz 160 deg; joints [1.674, 59.429, 11.397, -157.181, 72.229, 172.682]
  Set speed (17.8 mm/s)
  Call Extruder(818.31733)
  MoveL 4366 to (449.75, 460.76, 76) mm, rotated rx -180 ry 0 rz 160 deg; joints [1.396, 59.585, 11.023, -157.443, 71.992, 172.682]
  Set speed (17.8 mm/s)
  Call Extruder(825.68294)
  MoveL 4367 to (451.21, 458.96, 76) mm, rotated rx -180 ry 0 rz 160 deg; joints [1.133, 59.747, 10.634, -157.689, 71.749, 172.677]
  Set speed (17.8 mm/s)
  Call Extruder(833.12034)
  MoveL 4368 to (452.75, 457.2, 76) mm, rotated rx -180 ry 0 rz 160 deg; joints [0.877, 59.921, 10.218, -157.926, 71.492, 172.665]
  Set speed (17.8 mm/s)
  Call Extruder(840.50625)
  MoveL 4369 to (454.35, 455.5, 76) mm, rotated rx 180 ry 0 rz 160 deg; joints [0.633, 60.103, 9.784, -158.15, 71.227, 172.647]
  Set speed (17.8 mm/s)
  Call Extruder(848.01297)
  MoveL 4370 to (456.03, 453.84, 76) mm, rotated rx 180 ry 0 rz 160 deg; joints [0.395, 60.298, 9.321, -158.366, 70.948, 172.623]
  Set speed (17.8 mm/s)
  Call Extruder(855.45887)
  MoveL 4371 to (457.76, 452.25, 76) mm, rotated rx -180 ry 0 rz 160 deg; joints [0.169, 60.5, 8.841, -158.567, 70.661, 172.593]
  Set speed (17.8 mm/s)
  Call Extruder(862.99339)
  MoveL 4372 to (459.56, 450.71, 76) mm, rotated rx -180 ry 0 rz 160 deg; joints [-0.047, 60.715, 8.335, -158.757, 70.361, 172.556]
  Set speed (17.8 mm/s)
  Call Extruder(870.72631)
  MoveL 4373 to (461.48, 449.2, 76) mm, rotated rx -180 ry 0 rz 160 deg; joints [-0.257, 60.944, 7.796, -158.938, 70.044, 172.512]
  Set speed (17.8 mm/s)
  Call Extruder(877.33119)
  MoveL 4374 to (463.15, 447.97, 76) mm, rotated rx -180 ry 0 rz 160 deg; joints [-0.427, 61.147, 7.319, -159.082, 69.767, 172.47]
  Set speed (17.8 mm/s)
  Call Extruder(885.24688)
  MoveL 4375 to (465.22, 446.57, 76) mm, rotated rx 180 ry 0 rz 160 deg; joints [-0.618, 61.399, 6.728, -159.239, 69.425, 172.412]
  Set speed (17.8 mm/s)
  Call Extruder(892.79616)
  MoveL 4376 to (467.24, 445.31, 76) mm, rotated rx -180 ry 0 rz 160 deg; joints [-0.789, 61.649, 6.146, -159.375, 69.091, 172.35]
  Set speed (17.8 mm/s)
  Call Extruder(900.23384)
  MoveL 4377 to (469.27, 444.14, 76) mm, rotated rx 180 ry 0 rz 160 deg; joints [-0.945, 61.903, 5.555, -159.495, 68.756, 172.283]
  Set speed (17.8 mm/s)
  Call Extruder(907.64070)
  MoveL 4378 to (471.33, 443.05, 76) mm, rotated rx -180 ry 0 rz 160 deg; joints [-1.088, 62.164, 4.951, -159.601, 68.414, 172.21]
  Set speed (17.8 mm/s)
  Call Extruder(915.08085)
  MoveL 4379 to (473.45, 442.04, 76) mm, rotated rx -180 ry 0 rz 160 deg; joints [-1.22, 62.434, 4.328, -159.693, 68.065, 172.13]
  Set speed (17.8 mm/s)
  Call Extruder(922.58158)
  MoveL 4380 to (475.62, 441.09, 76) mm, rotated rx 180 ry 0 rz 160 deg; joints [-1.341, 62.713, 3.685, -159.771, 67.708, 172.043]
  Set speed (17.8 mm/s)
  Call Extruder(929.94206)
  MoveL 4381 to (477.77, 440.24, 76) mm, rotated rx 180 ry 0 rz 160 deg; joints [-1.449, 62.995, 3.04, -159.834, 67.352, 171.951]
  Set speed (17.8 mm/s)
  Call Extruder(937.46865)
  MoveL 4382 to (480.01, 439.46, 76) mm, rotated rx -180 ry 0 rz 160 deg; joints [-1.546, 63.289, 2.367, -159.883, 66.983, 171.85]
  Set speed (17.8 mm/s)
  Call Extruder(944.86910)
  MoveL 4383 to (482.24, 438.77, 76) mm, rotated rx -180 ry 0 rz 160 deg; joints [-1.629, 63.585, 1.693, -159.918, 66.615, 171.744]
  Call Extruder(952.37385)
  MoveL 4384 to (484.52, 438.15, 76) mm, rotated rx -180 ry 0 rz 160 deg; joints [-1.702, 63.892, 0.997, -159.938, 66.239, 171.629]
  Set speed (17.8 mm/s)
  Call Extruder(959.72112)
  MoveL 4385 to (486.78, 437.63, 76) mm, rotated rx 180 ry 0 rz 160 deg; joints [-1.762, 64.198, 0.304, -159.944, 65.868, 171.511]
  Set speed (17.8 mm/s)
  Call Extruder(967.12100)
  MoveL 4386 to (489.07, 437.19, 76) mm, rotated rx 180 ry 0 rz 160 deg; joints [-1.81, 64.512, -0.404, -159.936, 65.49, 171.384]
  Set speed (17.8 mm/s)
  Call Extruder(974.49648)
  MoveL 4387 to (491.37, 436.83, 76) mm, rotated rx 180 ry 0 rz 160 deg; joints [-1.847, 64.83, -1.118, -159.913, 65.112, 171.251]
  Set speed (17.8 mm/s)
  Call Extruder(982.06797)
  MoveL 4388 to (493.73, 436.55, 76) mm, rotated rx -180 ry 0 rz 160 deg; joints [-1.873, 65.162, -1.861, -159.875, 64.722, 171.107]
  Set speed (17.8 mm/s)
  Call Extruder(989.43989)
  MoveL 4389 to (496.05, 436.37, 76) mm, rotated rx 180 ry 0 rz 160 deg; joints [-1.887, 65.49, -2.593, -159.825, 64.34, 170.959]
  Set speed (17.8 mm/s)
  Call Extruder(997.05372)
  MoveL 4390 to (498.45, 436.26, 76) mm, rotated rx 180 ry 0 rz 160 deg; joints [-1.891, 65.833, -3.357, -159.757, 63.945, 170.799]
  Call Extruder(1004.41970)
  MoveL 4391 to (500.77, 436.25, 76) mm, rotated rx -180 ry 0 rz 160 deg; joints [-1.883, 66.169, -4.103, -159.679, 63.562, 170.637]
  Call Extruder(1011.93804)
  MoveL 4392 to (503.14, 436.32, 76) mm, rotated rx 180 ry 0 rz 160 deg; joints [-1.864, 66.516, -4.87, -159.584, 63.172, 170.464]
  Call Extruder(1019.31141)
  MoveL 4393 to (505.46, 436.48, 76) mm, rotated rx 180 ry 0 rz 160 deg; joints [-1.834, 66.86, -5.627, -159.478, 62.789, 170.287]
  Set speed (17.8 mm/s)
  Call Extruder(1026.82298)
  MoveL 4394 to (507.82, 436.73, 76) mm, rotated rx 180 ry 0 rz 160 deg; joints [-1.794, 67.212, -6.402, -159.356, 62.4, 170.099]
  Call Extruder(1034.19171)
  MoveL 4395 to (510.12, 437.05, 76) mm, rotated rx 180 ry 0 rz 160 deg; joints [-1.744, 67.561, -7.166, -159.224, 62.021, 169.907]
  Set speed (17.8 mm/s)
  Call Extruder(1041.62991)
  MoveL 4396 to (512.43, 437.47, 76) mm, rotated rx 180 ry 0 rz 160 deg; joints [-1.684, 67.915, -7.939, -159.077, 61.639, 169.706]
  Set speed (17.8 mm/s)
  Call Extruder(1048.50573)
  MoveL 4397 to (514.54, 437.93, 76) mm, rotated rx 180 ry 0 rz 160 deg; joints [-1.62, 68.243, -8.655, -158.929, 61.289, 169.514]
  Set speed (17.8 mm/s)
  Call Extruder(1056.45790)
  MoveL 4398 to (516.97, 438.55, 76) mm, rotated rx -180 ry 0 rz 160 deg; joints [-1.535, 68.624, -9.483, -158.745, 60.888, 169.284]
  Set speed (17.8 mm/s)
  Call Extruder(1063.96989)
  MoveL 4399 to (519.24, 439.22, 76) mm, rotated rx 180 ry 0 rz 160 deg; joints [-1.446, 68.986, -10.266, -158.558, 60.512, 169.059]
  Call Extruder(1071.32424)
  MoveL 4400 to (521.44, 439.96, 76) mm, rotated rx -180 ry 0 rz 160 deg; joints [-1.349, 69.34, -11.031, -158.363, 60.149, 168.831]
  Set speed (17.8 mm/s)
  Call Extruder(1078.74171)
  MoveL 4401 to (523.63, 440.79, 76) mm, rotated rx -180 ry 0 rz 160 deg; joints [-1.243, 69.697, -11.8, -158.154, 59.786, 168.594]
  Set speed (17.8 mm/s)
  Call Extruder(1086.38142)
  MoveL 4402 to (525.85, 441.72, 76) mm, rotated rx -180 ry 0 rz 160 deg; joints [-1.124, 70.064, -12.589, -157.927, 59.419, 168.343]
  Set speed (17.8 mm/s)
  Call Extruder(1093.75963)
  MoveL 4403 to (527.96, 442.7, 76) mm, rotated rx 180 ry 0 rz 160 deg; joints [-1.001, 70.418, -13.348, -157.696, 59.069, 168.094]
  Set speed (17.8 mm/s)
  Call Extruder(1101.28137)
  MoveL 4404 to (530.07, 443.78, 76) mm, rotated rx 180 ry 0 rz 160 deg; joints [-0.868, 70.777, -14.116, -157.45, 58.719, 167.833]
  Call Extruder(1108.72939)
  MoveL 4405 to (532.12, 444.92, 76) mm, rotated rx -180 ry 0 rz 160 deg; joints [-0.728, 71.131, -14.871, -157.195, 58.379, 167.568]
  Set speed (17.8 mm/s)
  Call Extruder(1116.07726)
  MoveL 4406 to (534.1, 446.13, 76) mm, rotated rx -180 ry 0 rz 160 deg; joints [-0.583, 71.477, -15.608, -156.933, 58.051, 167.301]
  Set speed (17.8 mm/s)
  Call Extruder(1123.61201)
  MoveL 4407 to (536.08, 447.44, 76) mm, rotated rx -180 ry 0 rz 160 deg; joints [-0.426, 71.829, -16.355, -156.655, 57.722, 167.021]
  Set speed (17.8 mm/s)
  Call Extruder(1130.97148)
  MoveL 4408 to (537.97, 448.79, 76) mm, rotated rx 180 ry 0 rz 160 deg; joints [-0.266, 72.17, -17.077, -156.374, 57.409, 166.742]
  Call Extruder(1138.30716)
  MoveL 4409 to (539.8, 450.19, 76) mm, rotated rx -180 ry 0 rz 160 deg; joints [-0.099, 72.505, -17.786, -156.085, 57.106, 166.459]
  Call Extruder(1145.86267)
  MoveL 4410 to (541.64, 451.72, 76) mm, rotated rx -180 ry 0 rz 160 deg; joints [0.079, 72.846, -18.504, -155.778, 56.803, 166.163]
  Call Extruder(1153.39466)
  MoveL 4411 to (543.4, 453.3, 76) mm, rotated rx -180 ry 0 rz 160 deg; joints [0.263, 73.179, -19.207, -155.464, 56.511, 165.863]
  Call Extruder(1160.78451)
  MoveL 4412 to (545.08, 454.92, 76) mm, rotated rx 180 ry 0 rz 160 deg; joints [0.449, 73.502, -19.884, -155.149, 56.234, 165.565]
  Set speed (17.8 mm/s)
  Call Extruder(1164.89480)
  MoveL 4413 to (545.99, 455.84, 76) mm, rotated rx -180 ry 0 rz 160 deg; joints [0.555, 73.678, -20.254, -154.97, 56.086, 165.397]
  Call Extruder(1168.96404)
  MoveL 4414 to (546.87, 456.78, 76) mm, rotated rx -180 ry 0 rz 160 deg; joints [0.662, 73.85, -20.615, -154.791, 55.942, 165.231]
  Call Extruder(1173.12616)
  MoveL 4415 to (547.75, 457.75, 76) mm, rotated rx -180 ry 0 rz 160 deg; joints [0.773, 74.025, -20.981, -154.607, 55.797, 165.06]
  Set speed (17.8 mm/s)
  Call Extruder(1177.35810)
  MoveL 4416 to (548.62, 458.76, 76) mm, rotated rx -180 ry 0 rz 160 deg; joints [0.888, 74.199, -21.346, -154.417, 55.655, 164.885]
  Set speed (17.8 mm/s)
  Call Extruder(1181.34921)
  MoveL 4417 to (549.42, 459.72, 76) mm, rotated rx 180 ry 0 rz 160 deg; joints [0.997, 74.362, -21.686, -154.236, 55.524, 164.719]
  Set speed (17.8 mm/s)
  Call Extruder(1185.51815)
  MoveL 4418 to (550.24, 460.75, 76) mm, rotated rx -180 ry 0 rz 160 deg; joints [1.114, 74.529, -22.035, -154.045, 55.391, 164.546]
  Set speed (17.8 mm/s)
  Call Extruder(1189.68667)
  MoveL 4419 to (551.04, 461.8, 76) mm, rotated rx 180 ry 0 rz 160 deg; joints [1.231, 74.694, -22.379, -153.853, 55.262, 164.372]
  Set speed (17.8 mm/s)
  Call Extruder(1193.33244)
  MoveL 4420 to (551.72, 462.72, 76) mm, rotated rx 180 ry 0 rz 160 deg; joints [1.335, 74.836, -22.674, -153.684, 55.152, 164.22]
  Call Extruder(1197.96344)
  MoveL 4421 to (552.56, 463.91, 76) mm, rotated rx 180 ry 0 rz 160 deg; joints [1.469, 75.013, -23.043, -153.467, 55.017, 164.026]
  Set speed (17.8 mm/s)
  Call Extruder(1202.14417)
  MoveL 4422 to (553.3, 465.01, 76) mm, rotated rx -180 ry 0 rz 160 deg; joints [1.592, 75.169, -23.368, -153.27, 54.9, 163.851]
  Call Extruder(1206.24286)
  MoveL 4423 to (553.99, 466.1, 76) mm, rotated rx -180 ry 0 rz 160 deg; joints [1.713, 75.319, -23.681, -153.076, 54.789, 163.679]
  Set speed (17.8 mm/s)
  Call Extruder(1210.39491)
  MoveL 4424 to (554.68, 467.21, 76) mm, rotated rx 180 ry 0 rz 160 deg; joints [1.838, 75.468, -23.99, -152.878, 54.682, 163.505]
  Set speed (17.8 mm/s)
  Call Extruder(1214.46185)
  MoveL 4425 to (555.32, 468.32, 76) mm, rotated rx -180 ry 0 rz 160 deg; joints [1.961, 75.611, -24.287, -152.684, 54.58, 163.335]
  Set speed (17.8 mm/s)
  Call Extruder(1218.61208)
  MoveL 4426 to (555.96, 469.46, 76) mm, rotated rx -180 ry 0 rz 160 deg; joints [2.087, 75.754, -24.582, -152.484, 54.481, 163.162]
  Set speed (17.8 mm/s)
  Call Extruder(1222.76319)
  MoveL 4427 to (556.58, 470.61, 76) mm, rotated rx 180 ry 0 rz 160 deg; joints [2.215, 75.893, -24.871, -152.284, 54.386, 162.99]
  Set speed (17.8 mm/s)
  Call Extruder(1226.92930)
  MoveL 4428 to (557.17, 471.78, 76) mm, rotated rx 180 ry 0 rz 160 deg; joints [2.345, 76.029, -25.153, -152.083, 54.295, 162.817]
  Set speed (17.8 mm/s)
  Call Extruder(1232.18940)
  MoveL 4429 to (557.89, 473.28, 76) mm, rotated rx -180 ry 0 rz 160 deg; joints [2.51, 76.196, -25.497, -151.829, 54.187, 162.6]
  Call Extruder(1235.16893)
  MoveL 4430 to (558.27, 474.13, 76) mm, rotated rx -180 ry 0 rz 160 deg; joints [2.605, 76.286, -25.685, -151.684, 54.13, 162.479]
  Set speed (17.8 mm/s)
  Call Extruder(1243.08646)
  MoveL 4431 to (559.24, 476.43, 76) mm, rotated rx 180 ry 0 rz 160 deg; joints [2.858, 76.52, -26.166, -151.3, 53.989, 162.157]
  Set speed (17.8 mm/s)
  Call Extruder(1247.69393)
  MoveL 4432 to (559.75, 477.79, 76) mm, rotated rx 180 ry 0 rz 160 deg; joints [3.008, 76.647, -26.43, -151.076, 53.915, 161.973]
  Set speed (17.8 mm/s)
  Call Extruder(1251.73348)
  MoveL 4433 to (560.19, 478.98, 76) mm, rotated rx 180 ry 0 rz 160 deg; joints [3.139, 76.757, -26.657, -150.881, 53.854, 161.811]
  Set speed (17.8 mm/s)
  Call Extruder(1255.94998)
  MoveL 4434 to (560.61, 480.24, 76) mm, rotated rx 180 ry 0 rz 160 deg; joints [3.277, 76.865, -26.879, -150.677, 53.798, 161.646]
  Set speed (17.8 mm/s)
  Call Extruder(1260.23449)
  MoveL 4435 to (561.02, 481.53, 76) mm, rotated rx -180 ry 0 rz 160 deg; joints [3.419, 76.972, -27.101, -150.47, 53.743, 161.478]
  Call Extruder(1264.24692)
  MoveL 4436 to (561.37, 482.74, 76) mm, rotated rx -180 ry 0 rz 160 deg; joints [3.552, 77.067, -27.294, -150.277, 53.699, 161.325]
  Set speed (17.8 mm/s)
  Call Extruder(1268.19947)
  MoveL 4437 to (561.7, 483.94, 76) mm, rotated rx -180 ry 0 rz 160 deg; joints [3.684, 77.157, -27.481, -150.087, 53.658, 161.174]
  Call Extruder(1272.53103)
  MoveL 4438 to (562.02, 485.26, 76) mm, rotated rx 180 ry 0 rz 160 deg; joints [3.829, 77.249, -27.67, -149.881, 53.621, 161.012]
  Call Extruder(1276.62332)
  MoveL 4439 to (562.32, 486.52, 76) mm, rotated rx -180 ry 0 rz 160 deg; joints [3.967, 77.334, -27.844, -149.686, 53.589, 160.86]
  Set speed (17.8 mm/s)
  Call Extruder(1284.91925)
  MoveL 4440 to (562.82, 489.08, 76) mm, rotated rx 180 ry 0 rz 160 deg; joints [4.248, 77.488, -28.162, -149.294, 53.541, 160.561]
  Set speed (17.8 mm/s)
  Call Extruder(1293.13511)
  MoveL 4441 to (563.21, 491.64, 76) mm, rotated rx -180 ry 0 rz 160 deg; joints [4.53, 77.622, -28.436, -148.911, 53.515, 160.275]
  Set speed (17.8 mm/s)
  Call Extruder(1301.57135)
  MoveL 4442 to (563.5, 494.29, 76) mm, rotated rx 180 ry 0 rz 160 deg; joints [4.82, 77.739, -28.676, -148.524, 53.508, 159.993]
  Set speed (17.8 mm/s)
  Call Extruder(1309.73815)
  MoveL 4443 to (563.68, 496.86, 76) mm, rotated rx -180 ry 0 rz 160 deg; joints [5.104, 77.831, -28.865, -148.155, 53.523, 159.734]
  Call Extruder(1318.02234)
  MoveL 4444 to (563.75, 499.47, 76) mm, rotated rx 180 ry 0 rz 160 deg; joints [5.392, 77.904, -29.014, -147.789, 53.559, 159.484]
  Set speed (17.8 mm/s)
  Call Extruder(1326.17519)
  MoveL 4445 to (563.72, 502.04, 76) mm, rotated rx 180 ry 0 rz 160 deg; joints [5.677, 77.954, -29.117, -147.437, 53.615, 159.252]
  Set speed (17.8 mm/s)
  Call Extruder(1334.55009)
  MoveL 4446 to (563.58, 504.67, 76) mm, rotated rx 180 ry 0 rz 160 deg; joints [5.97, 77.984, -29.179, -147.085, 53.693, 159.029]
  Set speed (17.8 mm/s)
  Call Extruder(1342.74780)
  MoveL 4447 to (563.34, 507.25, 76) mm, rotated rx -180 ry 0 rz 160 deg; joints [6.257, 77.992, -29.195, -146.749, 53.789, 158.827]
  Set speed (17.8 mm/s)
  Call Extruder(1351.18537)
  MoveL 4448 to (562.99, 509.89, 76) mm, rotated rx 180 ry 0 rz 160 deg; joints [6.553, 77.978, -29.166, -146.414, 53.909, 158.636]
  Set speed (17.8 mm/s)
  Call Extruder(1359.27195)
  MoveL 4449 to (562.54, 512.4, 76) mm, rotated rx -180 ry 0 rz 160 deg; joints [6.836, 77.943, -29.094, -146.103, 54.042, 158.469]
  Call Extruder(1367.68335)
  MoveL 4450 to (561.97, 514.99, 76) mm, rotated rx -180 ry 0 rz 160 deg; joints [7.129, 77.885, -28.976, -145.791, 54.201, 158.314]
  Set speed (17.8 mm/s)
  Call Extruder(1371.79812)
  MoveL 4451 to (561.65, 516.24, 76) mm, rotated rx -180 ry 0 rz 160 deg; joints [7.272, 77.847, -28.898, -145.643, 54.287, 158.246]
  Set speed (17.8 mm/s)
  Call Extruder(1376.06816)
  MoveL 4452 to (561.3, 517.54, 76) mm, rotated rx -180 ry 0 rz 160 deg; joints [7.42, 77.805, -28.813, -145.491, 54.378, 158.178]
  Call Extruder(1380.11840)
  MoveL 4453 to (560.93, 518.76, 76) mm, rotated rx -180 ry 0 rz 160 deg; joints [7.561, 77.758, -28.715, -145.352, 54.471, 158.12]
  Set speed (17.8 mm/s)
  Call Extruder(1384.27979)
  MoveL 4454 to (560.54, 520.01, 76) mm, rotated rx -180 ry 0 rz 160 deg; joints [7.704, 77.706, -28.609, -145.21, 54.569, 158.062]
  Set speed (17.8 mm/s)
  Call Extruder(1392.60332)
  MoveL 4455 to (559.66, 522.49, 76) mm, rotated rx -180 ry 0 rz 160 deg; joints [7.991, 77.585, -28.36, -144.937, 54.781, 157.964]
  Set speed (17.8 mm/s)
  Call Extruder(1396.62755)
  MoveL 4456 to (559.19, 523.67, 76) mm, rotated rx 180 ry 0 rz 160 deg; joints [8.128, 77.518, -28.222, -144.809, 54.891, 157.924]
  Set speed (17.8 mm/s)
  Call Extruder(1400.85555)
  MoveL 4457 to (558.69, 524.9, 76) mm, rotated rx -180 ry 0 rz 160 deg; joints [8.272, 77.445, -28.072, -144.677, 55.008, 157.884]
  Set speed (17.8 mm/s)
  Call Extruder(1404.90710)
  MoveL 4458 to (558.18, 526.07, 76) mm, rotated rx -180 ry 0 rz 160 deg; joints [8.41, 77.368, -27.913, -144.555, 55.126, 157.853]
  Set speed (17.8 mm/s)
  Call Extruder(1409.02573)
  MoveL 4459 to (557.64, 527.25, 76) mm, rotated rx 180 ry 0 rz 160 deg; joints [8.549, 77.287, -27.747, -144.433, 55.248, 157.824]
  Set speed (17.8 mm/s)
  Call Extruder(1412.20155)
  MoveL 4460 to (557.21, 528.15, 76) mm, rotated rx 180 ry 0 rz 160 deg; joints [8.656, 77.221, -27.612, -144.34, 55.345, 157.804]
  Set speed (17.8 mm/s)
  Call Extruder(1419.40978)
  MoveL 4461 to (556.17, 530.17, 76) mm, rotated rx -180 ry 0 rz 160 deg; joints [8.898, 77.061, -27.282, -144.137, 55.574, 157.771]
  Set speed (17.8 mm/s)
  Call Extruder(1425.50427)
  MoveL 4462 to (555.23, 531.85, 76) mm, rotated rx -180 ry 0 rz 160 deg; joints [9.1, 76.913, -26.977, -143.973, 55.778, 157.755]
  Set speed (17.8 mm/s)
  Call Extruder(1430.48736)
  MoveL 4463 to (554.43, 533.2, 76) mm, rotated rx 180 ry 0 rz 160 deg; joints [9.264, 76.785, -26.715, -143.843, 55.949, 157.748]
  Call Extruder(1433.77106)
  MoveL 4464 to (553.88, 534.08, 76) mm, rotated rx -180 ry 0 rz 160 deg; joints [9.371, 76.698, -26.534, -143.761, 56.065, 157.747]
  Set speed (17.8 mm/s)
  Call Extruder(1437.92313)
  MoveL 4465 to (553.17, 535.18, 76) mm, rotated rx -180 ry 0 rz 160 deg; joints [9.506, 76.584, -26.299, -143.659, 56.214, 157.75]
  Call Extruder(1442.07224)
  MoveL 4466 to (552.44, 536.26, 76) mm, rotated rx -180 ry 0 rz 160 deg; joints [9.64, 76.466, -26.055, -143.559, 56.366, 157.757]
  Set speed (17.8 mm/s)
  Call Extruder(1446.19581)
  MoveL 4467 to (551.69, 537.33, 76) mm, rotated rx -180 ry 0 rz 160 deg; joints [9.772, 76.344, -25.803, -143.464, 56.52, 157.768]
  Set speed (17.8 mm/s)
  Call Extruder(1450.31670)
  MoveL 4468 to (550.92, 538.37, 76) mm, rotated rx -180 ry 0 rz 160 deg; joints [9.903, 76.219, -25.545, -143.371, 56.677, 157.784]
  Call Extruder(1454.42371)
  MoveL 4469 to (550.13, 539.4, 76) mm, rotated rx -180 ry 0 rz 160 deg; joints [10.033, 76.09, -25.279, -143.281, 56.836, 157.803]
  Set speed (17.8 mm/s)
  Call Extruder(1458.66116)
  MoveL 4470 to (549.29, 540.44, 76) mm, rotated rx -180 ry 0 rz 160 deg; joints [10.165, 75.953, -24.996, -143.192, 57.003, 157.828]
  Set speed (17.8 mm/s)
  Call Extruder(1462.73359)
  MoveL 4471 to (548.47, 541.42, 76) mm, rotated rx -180 ry 0 rz 160 deg; joints [10.292, 75.818, -24.716, -143.109, 57.167, 157.855]
  Set speed (17.8 mm/s)
  Call Extruder(1466.85986)
  MoveL 4472 to (547.61, 542.4, 76) mm, rotated rx 180 ry 0 rz 160 deg; joints [10.418, 75.678, -24.425, -143.027, 57.335, 157.887]
  Set speed (17.8 mm/s)
  Call Extruder(1470.98406)
  MoveL 4473 to (546.74, 543.37, 76) mm, rotated rx 180 ry 0 rz 160 deg; joints [10.544, 75.535, -24.127, -142.949, 57.505, 157.923]
  Set speed (17.8 mm/s)
  Call Extruder(1475.16865)
  MoveL 4474 to (545.83, 544.32, 76) mm, rotated rx -180 ry 0 rz 160 deg; joints [10.67, 75.386, -23.818, -142.872, 57.68, 157.964]
  Call Extruder(1479.42791)
  MoveL 4475 to (544.88, 545.28, 76) mm, rotated rx -180 ry 0 rz 160 deg; joints [10.797, 75.231, -23.496, -142.796, 57.861, 158.009]
  Set speed (17.8 mm/s)
  Call Extruder(1483.45677)
  MoveL 4476 to (543.97, 546.16, 76) mm, rotated rx 180 ry 0 rz 160 deg; joints [10.915, 75.081, -23.185, -142.728, 58.034, 158.055]
  Set speed (17.8 mm/s)
  Call Extruder(1488.26441)
  MoveL 4477 to (542.87, 547.2, 76) mm, rotated rx 180 ry 0 rz 160 deg; joints [11.055, 74.899, -22.807, -142.649, 58.242, 158.115]
  Set speed (17.8 mm/s)
  Call Extruder(1491.72727)
  MoveL 4478 to (542.05, 547.92, 76) mm, rotated rx 180 ry 0 rz 160 deg; joints [11.154, 74.766, -22.528, -142.595, 58.395, 158.162]
  Set speed (17.8 mm/s)
  Call Extruder(1495.81553)
  MoveL 4479 to (541.07, 548.76, 76) mm, rotated rx 180 ry 0 rz 160 deg; joints [11.27, 74.605, -22.193, -142.534, 58.576, 158.22]
  Set speed (17.8 mm/s)
  Call Extruder(1499.94239)
  MoveL 4480 to (540.07, 549.59, 76) mm, rotated rx 180 ry 0 rz 160 deg; joints [11.386, 74.441, -21.851, -142.474, 58.76, 158.281]
  Call Extruder(1504.14210)
  MoveL 4481 to (539.03, 550.41, 76) mm, rotated rx -180 ry 0 rz 160 deg; joints [11.502, 74.271, -21.496, -142.416, 58.95, 158.348]
  Call Extruder(1508.28334)
  MoveL 4482 to (537.99, 551.2, 76) mm, rotated rx -180 ry 0 rz 160 deg; joints [11.615, 74.101, -21.14, -142.362, 59.139, 158.417]
  Set speed (17.8 mm/s)
  Call Extruder(1512.37382)
  MoveL 4483 to (536.95, 551.96, 76) mm, rotated rx -180 ry 0 rz 160 deg; joints [11.725, 73.93, -20.783, -142.311, 59.326, 158.489]
  Call Extruder(1516.58878)
  MoveL 4484 to (535.86, 552.72, 76) mm, rotated rx -180 ry 0 rz 160 deg; joints [11.836, 73.753, -20.412, -142.26, 59.521, 158.565]
  Set speed (17.8 mm/s)
  Call Extruder(1520.63560)
  MoveL 4485 to (534.8, 553.42, 76) mm, rotated rx 180 ry 0 rz 160 deg; joints [11.942, 73.58, -20.049, -142.215, 59.709, 158.643]
  Set speed (17.8 mm/s)
  Call Extruder(1524.77402)
  MoveL 4486 to (533.7, 554.12, 76) mm, rotated rx 180 ry 0 rz 160 deg; joints [12.048, 73.402, -19.674, -142.17, 59.903, 158.724]
  Set speed (17.8 mm/s)
  Call Extruder(1528.91674)
  MoveL 4487 to (532.58, 554.8, 76) mm, rotated rx -180 ry 0 rz 160 deg; joints [12.152, 73.221, -19.295, -142.129, 60.098, 158.809]
  Call Extruder(1532.40771)
  MoveL 4488 to (531.63, 555.36, 76) mm, rotated rx 180 ry 0 rz 160 deg; joints [12.238, 73.067, -18.971, -142.096, 60.263, 158.883]
  Set speed (17.8 mm/s)
  Call Extruder(1537.15648)
  MoveL 4489 to (530.33, 556.09, 76) mm, rotated rx -180 ry 0 rz 160 deg; joints [12.354, 72.856, -18.527, -142.053, 60.488, 158.987]
  Set speed (17.8 mm/s)
  Call Extruder(1542.56225)
  MoveL 4490 to (528.82, 556.87, 76) mm, rotated rx -180 ry 0 rz 160 deg; joints [12.482, 72.613, -18.015, -142.009, 60.746, 159.11]
  Set speed (17.8 mm/s)
  Call Extruder(1545.53718)
  MoveL 4491 to (527.98, 557.29, 76) mm, rotated rx 180 ry 0 rz 160 deg; joints [12.55, 72.478, -17.73, -141.987, 60.889, 159.18]
  Set speed (17.8 mm/s)
  Call Extruder(1549.74626)
  MoveL 4492 to (526.78, 557.86, 76) mm, rotated rx 180 ry 0 rz 160 deg; joints [12.647, 72.287, -17.324, -141.958, 61.091, 159.28]
  Set speed (17.8 mm/s)
  Call Extruder(1553.84245)
  MoveL 4493 to (525.6, 558.38, 76) mm, rotated rx 180 ry 0 rz 160 deg; joints [12.737, 72.098, -16.925, -141.932, 61.289, 159.382]
  Set speed (17.8 mm/s)
  Call Extruder(1558.12642)
  MoveL 4494 to (524.36, 558.92, 76) mm, rotated rx 180 ry 0 rz 160 deg; joints [12.831, 71.901, -16.508, -141.907, 61.496, 159.489]
  Set speed (17.8 mm/s)
  Call Extruder(1562.11133)
  MoveL 4495 to (523.2, 559.38, 76) mm, rotated rx -180 ry 0 rz 160 deg; joints [12.915, 71.715, -16.113, -141.887, 61.689, 159.593]
  Call Extruder(1566.07420)
  MoveL 4496 to (522.03, 559.83, 76) mm, rotated rx -180 ry 0 rz 160 deg; joints [12.997, 71.53, -15.721, -141.868, 61.881, 159.697]
  Set speed (17.8 mm/s)
  Call Extruder(1570.46138)
  MoveL 4497 to (520.73, 560.29, 76) mm, rotated rx 180 ry 0 rz 160 deg; joints [13.085, 71.324, -15.282, -141.851, 62.094, 159.816]
  Call Extruder(0.00000)
  Set speed (17.8 mm/s)
  Call Extruder(4.12610)
  MoveL 4498 to (519.5, 560.7, 76) mm, rotated rx 180 ry 0 rz 160 deg; joints [13.166, 71.13, -14.869, -141.836, 62.294, 159.928]
  Call Extruder(8.21841)
  MoveL 4499 to (518.27, 561.08, 76) mm, rotated rx -180 ry 0 rz 160 deg; joints [13.243, 70.936, -14.455, -141.825, 62.494, 160.044]
  Call Extruder(12.21943)
  MoveL 4500 to (517.06, 561.43, 76) mm, rotated rx 180 ry 0 rz 160 deg; joints [13.318, 70.746, -14.051, -141.815, 62.688, 160.157]
  Set speed (17.8 mm/s)
  Call Extruder(15.97075)
  MoveL 4501 to (515.92, 561.73, 76) mm, rotated rx -180 ry 0 rz 160 deg; joints [13.384, 70.568, -13.668, -141.81, 62.87, 160.266]
  Set speed (17.8 mm/s)
  Call Extruder(20.60287)
  MoveL 4502 to (514.5, 562.09, 76) mm, rotated rx -180 ry 0 rz 160 deg; joints [13.465, 70.347, -13.196, -141.804, 63.095, 160.402]
  Set speed (17.8 mm/s)
  Call Extruder(28.94362)
  MoveL 4503 to (511.93, 562.63, 76) mm, rotated rx -180 ry 0 rz 160 deg; joints [13.601, 69.947, -12.337, -141.803, 63.501, 160.655]
  Call Extruder(37.26252)
  MoveL 4504 to (509.35, 563.07, 76) mm, rotated rx -180 ry 0 rz 160 deg; joints [13.727, 69.547, -11.477, -141.811, 63.904, 160.914]
  Set speed (17.8 mm/s)
  Call Extruder(45.45413)
  MoveL 4505 to (506.78, 563.39, 76) mm, rotated rx 180 ry 0 rz 160 deg; joints [13.839, 69.152, -10.625, -141.83, 64.3, 161.176]
  Set speed (17.8 mm/s)
  Call Extruder(53.77869)
  MoveL 4506 to (504.17, 563.62, 76) mm, rotated rx -180 ry 0 rz 160 deg; joints [13.943, 68.751, -9.759, -141.859, 64.7, 161.449]
  Set speed (17.8 mm/s)
  Call Extruder(62.09329)
  MoveL 4507 to (501.55, 563.74, 76) mm, rotated rx 180 ry 0 rz 160 deg; joints [14.035, 68.352, -8.892, -141.897, 65.096, 161.726]
  Set speed (17.8 mm/s)
  Call Extruder(70.19803)
  MoveL 4508 to (499, 563.75, 76) mm, rotated rx 180 ry 0 rz 160 deg; joints [14.113, 67.965, -8.048, -141.945, 65.48, 162.002]
  Set speed (10.0 mm/s)
  MoveL 4509 to (499, 563.75, 80) mm, rotated rx 180 ry 0 rz 160 deg; joints [14.113, 67.303, -7.687, -141.86, 65.243, 161.798]
  Set speed (120.0 mm/s)
  MoveL 4510 to (498.98, 564.32, 80) mm, rotated rx -180 ry 0 rz 160 deg; joints [14.182, 67.323, -7.731, -141.781, 65.246, 161.752]
  Set speed (17.8 mm/s)
  Call Extruder(78.65912)
  MoveL 4511 to (496.31, 564.22, 80) mm, rotated rx -180 ry 0 rz 160 deg; joints [14.251, 66.918, -6.85, -141.843, 65.641, 162.044]
  Call Extruder(87.01307)
  MoveL 4512 to (493.68, 564.02, 80) mm, rotated rx 180 ry 0 rz 160 deg; joints [14.308, 66.52, -5.984, -141.913, 66.027, 162.337]
  Set speed (17.8 mm/s)
  Call Extruder(95.27848)
  MoveL 4513 to (491.09, 563.71, 80) mm, rotated rx 180 ry 0 rz 160 deg; joints [14.351, 66.13, -5.132, -141.994, 66.404, 162.63]
  Set speed (17.8 mm/s)
  Call Extruder(103.50288)
  MoveL 4514 to (488.52, 563.3, 80) mm, rotated rx 180 ry 0 rz 160 deg; joints [14.381, 65.746, -4.289, -142.085, 66.775, 162.925]
  Set speed (17.8 mm/s)
  Call Extruder(111.72871)
  MoveL 4515 to (485.97, 562.78, 80) mm, rotated rx -180 ry 0 rz 160 deg; joints [14.398, 65.365, -3.452, -142.187, 67.14, 163.223]
  Set speed (17.8 mm/s)
  Call Extruder(116.14240)
  MoveL 4516 to (484.62, 562.46, 80) mm, rotated rx -180 ry 0 rz 160 deg; joints [14.401, 65.163, -3.006, -142.246, 67.334, 163.384]
  Set speed (17.8 mm/s)
  Call Extruder(120.14437)
  MoveL 4517 to (483.39, 562.15, 80) mm, rotated rx 180 ry 0 rz 160 deg; joints [14.402, 64.981, -2.603, -142.302, 67.508, 163.529]
  Set speed (17.8 mm/s)
  Call Extruder(128.50645)
  MoveL 4518 to (480.85, 561.41, 80) mm, rotated rx 180 ry 0 rz 160 deg; joints [14.392, 64.604, -1.769, -142.427, 67.868, 163.836]
  Set speed (17.8 mm/s)
  Call Extruder(132.74356)
  MoveL 4519 to (479.58, 561, 80) mm, rotated rx 180 ry 0 rz 160 deg; joints [14.38, 64.415, -1.35, -142.496, 68.047, 163.991]
  Set speed (17.8 mm/s)
  Call Extruder(136.86269)
  MoveL 4520 to (478.35, 560.58, 80) mm, rotated rx 180 ry 0 rz 160 deg; joints [14.367, 64.233, -0.946, -142.563, 68.22, 164.142]
  Set speed (17.8 mm/s)
  Call Extruder(141.13162)
  MoveL 4521 to (477.09, 560.1, 80) mm, rotated rx -180 ry 0 rz 160 deg; joints [14.348, 64.047, -0.529, -142.638, 68.397, 164.299]
  Call Extruder(145.25206)
  MoveL 4522 to (475.87, 559.64, 80) mm, rotated rx 180 ry 0 rz 160 deg; joints [14.328, 63.868, -0.13, -142.712, 68.567, 164.451]
  Set speed (17.8 mm/s)
  Call Extruder(152.59090)
  MoveL 4523 to (473.74, 558.73, 80) mm, rotated rx 180 ry 0 rz 160 deg; joints [14.282, 63.553, 0.573, -142.851, 68.865, 164.721]
  Call Extruder(157.74871)
  MoveL 4524 to (472.26, 558.05, 80) mm, rotated rx 180 ry 0 rz 160 deg; joints [14.243, 63.336, 1.062, -142.954, 69.07, 164.91]
  Set speed (17.8 mm/s)
  Call Extruder(161.88389)
  MoveL 4525 to (471.09, 557.47, 80) mm, rotated rx 180 ry 0 rz 160 deg; joints [14.207, 63.163, 1.45, -143.041, 69.233, 165.062]
  Set speed (17.8 mm/s)
  Call Extruder(166.01958)
  MoveL 4526 to (469.93, 556.87, 80) mm, rotated rx 180 ry 0 rz 160 deg; joints [14.168, 62.992, 1.835, -143.13, 69.394, 165.214]
  Call Extruder(170.19263)
  MoveL 4527 to (468.77, 556.24, 80) mm, rotated rx -180 ry 0 rz 160 deg; joints [14.124, 62.822, 2.22, -143.223, 69.555, 165.367]
  Set speed (17.8 mm/s)
  Call Extruder(174.45081)
  MoveL 4528 to (467.6, 555.57, 80) mm, rotated rx 180 ry 0 rz 160 deg; joints [14.076, 62.649, 2.609, -143.32, 69.717, 165.522]
  Call Extruder(178.62103)
  MoveL 4529 to (466.47, 554.9, 80) mm, rotated rx 180 ry 0 rz 160 deg; joints [14.026, 62.483, 2.986, -143.419, 69.873, 165.674]
  Set speed (17.8 mm/s)
  Call Extruder(182.71282)
  MoveL 4530 to (465.37, 554.21, 80) mm, rotated rx -180 ry 0 rz 160 deg; joints [13.972, 62.322, 3.351, -143.519, 70.024, 165.823]
  Set speed (17.8 mm/s)
  Call Extruder(186.77434)
  MoveL 4531 to (464.3, 553.51, 80) mm, rotated rx -180 ry 0 rz 160 deg; joints [13.915, 62.164, 3.711, -143.62, 70.172, 165.97]
  Set speed (17.8 mm/s)
  Call Extruder(191.09286)
  MoveL 4532 to (463.17, 552.74, 80) mm, rotated rx -180 ry 0 rz 160 deg; joints [13.851, 61.998, 4.088, -143.732, 70.327, 166.125]
  Set speed (17.8 mm/s)
  Call Extruder(195.18876)
  MoveL 4533 to (462.12, 551.99, 80) mm, rotated rx -180 ry 0 rz 160 deg; joints [13.786, 61.843, 4.441, -143.84, 70.472, 166.272]
  Set speed (17.8 mm/s)
  Call Extruder(199.41312)
  MoveL 4534 to (461.04, 551.19, 80) mm, rotated rx 180 ry 0 rz 160 deg; joints [13.716, 61.685, 4.802, -143.955, 70.619, 166.423]
  Call Extruder(203.46791)
  MoveL 4535 to (460.03, 550.4, 80) mm, rotated rx -180 ry 0 rz 160 deg; joints [13.645, 61.536, 5.142, -144.068, 70.757, 166.567]
  Call Extruder(208.25564)
  MoveL 4536 to (458.86, 549.45, 80) mm, rotated rx 180 ry 0 rz 160 deg; joints [13.556, 61.363, 5.539, -144.205, 70.918, 166.735]
  Call Extruder(211.79522)
  MoveL 4537 to (458, 548.73, 80) mm, rotated rx 180 ry 0 rz 160 deg; joints [13.487, 61.238, 5.829, -144.308, 71.035, 166.859]
  Set speed (17.8 mm/s)
  Call Extruder(215.97853)
  MoveL 4538 to (457.01, 547.86, 80) mm, rotated rx -180 ry 0 rz 160 deg; joints [13.403, 61.091, 6.166, -144.434, 71.171, 167.005]
  Set speed (17.8 mm/s)
  Call Extruder(220.09580)
  MoveL 4539 to (456.05, 546.98, 80) mm, rotated rx 180 ry 0 rz 160 deg; joints [13.315, 60.949, 6.492, -144.56, 71.302, 167.147]
  Set speed (17.8 mm/s)
  Call Extruder(224.28444)
  MoveL 4540 to (455.09, 546.06, 80) mm, rotated rx 180 ry 0 rz 160 deg; joints [13.223, 60.808, 6.819, -144.691, 71.433, 167.291]
  Set speed (17.8 mm/s)
  Call Extruder(228.59232)
  MoveL 4541 to (454.13, 545.1, 80) mm, rotated rx 180 ry 0 rz 160 deg; joints [13.125, 60.665, 7.15, -144.829, 71.565, 167.437]
  Set speed (17.8 mm/s)
  Call Extruder(231.83869)
  MoveL 4542 to (453.42, 544.36, 80) mm, rotated rx -180 ry 0 rz 160 deg; joints [13.048, 60.559, 7.395, -144.935, 71.662, 167.547]
  Set speed (17.8 mm/s)
  Call Extruder(237.55472)
  MoveL 4543 to (452.19, 543.04, 80) mm, rotated rx -180 ry 0 rz 160 deg; joints [12.907, 60.377, 7.819, -145.125, 71.829, 167.738]
  Set speed (17.8 mm/s)
  Call Extruder(240.92059)
  MoveL 4544 to (451.49, 542.24, 80) mm, rotated rx -180 ry 0 rz 160 deg; joints [12.82, 60.272, 8.063, -145.24, 71.926, 167.849]
  Call Extruder(244.69429)
  MoveL 4545 to (450.71, 541.34, 80) mm, rotated rx -180 ry 0 rz 160 deg; joints [12.721, 60.156, 8.333, -145.371, 72.031, 167.973]
  Set speed (17.8 mm/s)
  Call Extruder(249.30558)
  MoveL 4546 to (449.79, 540.21, 80) mm, rotated rx -180 ry 0 rz 160 deg; joints [12.595, 60.018, 8.656, -145.534, 72.157, 168.123]
  Set speed (17.8 mm/s)
  Call Extruder(253.45473)
  MoveL 4547 to (448.98, 539.18, 80) mm, rotated rx -180 ry 0 rz 160 deg; joints [12.479, 59.896, 8.94, -145.683, 72.268, 168.256]
  Set speed (17.8 mm/s)
  Call Extruder(257.65012)
  MoveL 4548 to (448.18, 538.12, 80) mm, rotated rx -180 ry 0 rz 160 deg; joints [12.357, 59.776, 9.221, -145.837, 72.376, 168.389]
  Call Extruder(261.83096)
